gfCNCPoint4[3640] = {X 471.9427, Y 20.0094, Z -5.5000, A 0.000, B 0.000, C 0.000 }
gfCNCPoint4[3641] = {X 472.1592, Y 18.2535, Z -5.5000, A 0.000, B 0.000, C 0.000 }
gfCNCPoint4[3642] = {X 472.5540, Y 16.5288, Z -5.5000, A 0.000, B 0.000, C 0.000 }
gfCNCPoint4[3643] = {X 473.0727, Y 15.0578, Z -5.5000, A 0.000, B 0.000, C 0.000 }
gfCNCPoint4[3644] = {X 473.7721, Y 13.6637, Z -5.5000, A 0.000, B 0.000, C 0.000 }
gfCNCPoint4[3645] = {X 474.6410, Y 12.3684, Z -5.5000, A 0.000, B 0.000, C 0.000 }
gfCNCPoint4[3646] = {X 475.6658, Y 11.1925, Z -5.5000, A 0.000, B 0.000, C 0.000 }
gfCNCPoint4[3647] = {X 476.7434, Y 10.2234, Z -5.5000, A 0.000, B 0.000, C 0.000 }
gfCNCPoint4[3648] = {X 477.9268, Y 9.3867, Z -5.5000, A 0.000, B 0.000, C 0.000 }
gfCNCPoint4[3649] = {X 479.1997, Y 8.6938, Z -5.5000, A 0.000, B 0.000, C 0.000 }
gfCNCPoint4[3650] = {X 480.5449, Y 8.1544, Z -5.5000, A 0.000, B 0.000, C 0.000 }
gfCNCPoint4[3651] = {X 481.9438, Y 7.7756, Z -5.5000, A 0.000, B 0.000, C 0.000 }
gfCNCPoint4[3652] = {X 484.0949, Y 7.4404, Z -5.5000, A 0.000, B 0.000, C 0.000 }
gfCNCPoint4[3653] = {X 486.2687, Y 7.3224, Z -5.5000, A 0.000, B 0.000, C 0.000 }
gfCNCPoint4[3654] = {X 486.9707, Y 7.3102, Z -5.5000, A 0.000, B 0.000, C 0.000 }
gfCNCPoint4[3655] = {X 502.2122, Y 7.3103, Z -5.5000, A 0.000, B 0.000, C 0.000 }
gfCNCPoint4[3656] = {X 502.7439, Y 7.3144, Z -5.5000, A 0.000, B 0.000, C 0.000 }
gfCNCPoint4[3657] = {X 503.6982, Y 7.4166, Z -5.5000, A 0.000, B 0.000, C 0.000 }
gfCNCPoint4[3658] = {X 504.6139, Y 7.7042, Z -5.5000, A 0.000, B 0.000, C 0.000 }
gfCNCPoint4[3659] = {X 505.4552, Y 8.1661, Z -5.5000, A 0.000, B 0.000, C 0.000 }
gfCNCPoint4[3660] = {X 506.1895, Y 8.7843, Z -5.5000, A 0.000, B 0.000, C 0.000 }
gfCNCPoint4[3661] = {X 506.7880, Y 9.5346, Z -5.5000, A 0.000, B 0.000, C 0.000 }
gfCNCPoint4[3662] = {X 507.2274, Y 10.3879, Z -5.5000, A 0.000, B 0.000, C 0.000 }
gfCNCPoint4[3663] = {X 507.4825, Y 11.2663, Z -5.5000, A 0.000, B 0.000, C 0.000 }
gfCNCPoint4[3664] = {X 507.5685, Y 12.1769, Z -5.5000, A 0.000, B 0.000, C 0.000 }
gfCNCPoint4[3665] = {X 507.5683, Y 13.0237, Z -5.5000, A 0.000, B 0.000, C 0.000 }
gfCNCPoint4[3666] = {X 507.4609, Y 13.9970, Z -5.5000, A 0.000, B 0.000, C 0.000 }
gfCNCPoint4[3667] = {X 507.1614, Y 14.9292, Z -5.5000, A 0.000, B 0.000, C 0.000 }
gfCNCPoint4[3668] = {X 506.6818, Y 15.7829, Z -5.5000, A 0.000, B 0.000, C 0.000 }
gfCNCPoint4[3669] = {X 506.0415, Y 16.5237, Z -5.5000, A 0.000, B 0.000, C 0.000 }
gfCNCPoint4[3670] = {X 506.0414, Y 40.6631, Z -5.5000, A 0.000, B 0.000, C 0.000 }
gfCNCPoint4[3671] = {X 506.6823, Y 41.4045, Z -5.5000, A 0.000, B 0.000, C 0.000 }
gfCNCPoint4[3672] = {X 507.1621, Y 42.2591, Z -5.5000, A 0.000, B 0.000, C 0.000 }
gfCNCPoint4[3673] = {X 507.4614, Y 43.1923, Z -5.5000, A 0.000, B 0.000, C 0.000 }
gfCNCPoint4[3674] = {X 507.5683, Y 44.1665, Z -5.5000, A 0.000, B 0.000, C 0.000 }
gfCNCPoint4[3675] = {X 507.5685, Y 45.0000, Z -5.5000, A 0.000, B 0.000, C 0.000 }
gfCNCPoint4[3676] = {X 507.4747, Y 45.9520, Z -5.5000, A 0.000, B 0.000, C 0.000 }
gfCNCPoint4[3677] = {X 507.1970, Y 46.8675, Z -5.5000, A 0.000, B 0.000, C 0.000 }
gfCNCPoint4[3678] = {X 506.7461, Y 47.7112, Z -5.5000, A 0.000, B 0.000, C 0.000 }
gfCNCPoint4[3679] = {X 506.1392, Y 48.4507, Z -5.5000, A 0.000, B 0.000, C 0.000 }
gfCNCPoint4[3680] = {X 505.3997, Y 49.0576, Z -5.5000, A 0.000, B 0.000, C 0.000 }
gfCNCPoint4[3681] = {X 504.5560, Y 49.5085, Z -5.5000, A 0.000, B 0.000, C 0.000 }
gfCNCPoint4[3682] = {X 503.6405, Y 49.7862, Z -5.5000, A 0.000, B 0.000, C 0.000 }
gfCNCPoint4[3683] = {X 502.6885, Y 49.8800, Z -5.5000, A 0.000, B 0.000, C 0.000 }
gfCNCPoint4[3684] = {X 496.2450, Y 49.8800, Z -5.5000, A 0.000, B 0.000, C 0.000 }
gfCNCPoint4[3685] = {X 495.2220, Y 49.7716, Z -5.5000, A 0.000, B 0.000, C 0.000 }
gfCNCPoint4[3686] = {X 494.2445, Y 49.4511, Z -5.5000, A 0.000, B 0.000, C 0.000 }
gfCNCPoint4[3687] = {X 493.3559, Y 48.9328, Z -5.5000, A 0.000, B 0.000, C 0.000 }
gfCNCPoint4[3688] = {X 492.5956, Y 48.2398, Z -5.5000, A 0.000, B 0.000, C 0.000 }
gfCNCPoint4[3689] = {X 491.9976, Y 47.4028, Z -5.5000, A 0.000, B 0.000, C 0.000 }
gfCNCPoint4[3690] = {X 491.5882, Y 46.4590, Z -5.5000, A 0.000, B 0.000, C 0.000 }
gfCNCPoint4[3691] = {X 491.4241, Y 45.7570, Z -5.5000, A 0.000, B 0.000, C 0.000 }
gfCNCPoint4[3692] = {X 491.3652, Y 45.0385, Z -5.5000, A 0.000, B 0.000, C 0.000 }
gfCNCPoint4[3693] = {X 491.3655, Y 44.1416, Z -5.5000, A 0.000, B 0.000, C 0.000 }
gfCNCPoint4[3694] = {X 491.4758, Y 43.1751, Z -5.5000, A 0.000, B 0.000, C 0.000 }
gfCNCPoint4[3695] = {X 491.7756, Y 42.2497, Z -5.5000, A 0.000, B 0.000, C 0.000 }
gfCNCPoint4[3696] = {X 492.2530, Y 41.4020, Z -5.5000, A 0.000, B 0.000, C 0.000 }
gfCNCPoint4[3697] = {X 492.8890, Y 40.6660, Z -5.5000, A 0.000, B 0.000, C 0.000 }
gfCNCPoint4[3698] = {X 492.8890, Y 35.0338, Z -5.5000, A 0.000, B 0.000, C 0.000 }
gfCNCPoint4[3699] = {X 491.0668, Y 35.0338, Z -5.5000, A 0.000, B 0.000, C 0.000 }
gfCNCPoint4[3700] = {X 487.0440, Y 42.8709, Z -5.5000, A 0.000, B 0.000, C 0.000 }
gfCNCPoint4[3701] = {X 487.1810, Y 43.5116, Z -5.5000, A 0.000, B 0.000, C 0.000 }
gfCNCPoint4[3702] = {X 487.2308, Y 44.1648, Z -5.5000, A 0.000, B 0.000, C 0.000 }
gfCNCPoint4[3703] = {X 487.2310, Y 45.0000, Z -5.5000, A 0.000, B 0.000, C 0.000 }
gfCNCPoint4[3704] = {X 487.1749, Y 45.7380, Z -5.5000, A 0.000, B 0.000, C 0.000 }
gfCNCPoint4[3705] = {X 487.0078, Y 46.4590, Z -5.5000, A 0.000, B 0.000, C 0.000 }
gfCNCPoint4[3706] = {X 486.5939, Y 47.4110, Z -5.5000, A 0.000, B 0.000, C 0.000 }
gfCNCPoint4[3707] = {X 485.9879, Y 48.2538, Z -5.5000, A 0.000, B 0.000, C 0.000 }
gfCNCPoint4[3708] = {X 485.2175, Y 48.9494, Z -5.5000, A 0.000, B 0.000, C 0.000 }
gfCNCPoint4[3709] = {X 484.3173, Y 49.4663, Z -5.5000, A 0.000, B 0.000, C 0.000 }
gfCNCPoint4[3710] = {X 483.3557, Y 49.7755, Z -5.5000, A 0.000, B 0.000, C 0.000 }
gfCNCPoint4[3711] = {X 482.3510, Y 49.8800, Z -5.5000, A 0.000, B 0.000, C 0.000 }
gfCNCPoint4[3712] = {X 480.2695, Y 49.8800, Z -5.5000, A 0.000, B 0.000, C 0.000 }
gfCNCPoint4[3713] = {X 480.2695, Y 49.4000, Z -5.5000, A 0.000, B 0.000, C 0.000 }
gfCNCPoint4[3714] = {X 475.7650, Y 49.4000, Z -5.5000, A 0.000, B 0.000, C 0.000 }
gfCNCPoint4[3715] = {X 474.7859, Y 49.2897, Z -5.5000, A 0.000, B 0.000, C 0.000 }
gfCNCPoint4[3716] = {X 473.8559, Y 48.9643, Z -5.5000, A 0.000, B 0.000, C 0.000 }
gfCNCPoint4[3717] = {X 473.0216, Y 48.4401, Z -5.5000, A 0.000, B 0.000, C 0.000 }
gfCNCPoint4[3718] = {X 472.3249, Y 47.7434, Z -5.5000, A 0.000, B 0.000, C 0.000 }
gfCNCPoint4[3719] = {X 471.8007, Y 46.9091, Z -5.5000, A 0.000, B 0.000, C 0.000 }
gfCNCPoint4[3720] = {X 471.4753, Y 45.9791, Z -5.5000, A 0.000, B 0.000, C 0.000 }
gfCNCPoint4[3721] = {X 471.3650, Y 45.0000, Z -5.5000, A 0.000, B 0.000, C 0.000 }
gfCNCPoint4[3722] = {X 471.3654, Y 44.1483, Z -5.5000, A 0.000, B 0.000, C 0.000 }
gfCNCPoint4[3723] = {X 471.4638, Y 43.2816, Z -5.5000, A 0.000, B 0.000, C 0.000 }
gfCNCPoint4[3724] = {X 471.7311, Y 42.4514, Z -5.5000, A 0.000, B 0.000, C 0.000 }
gfCNCPoint4[3725] = {X 472.1570, Y 41.6903, Z -5.5000, A 0.000, B 0.000, C 0.000 }
gfCNCPoint4[3726] = {X 472.7247, Y 41.0281, Z -5.5000, A 0.000, B 0.000, C 0.000 }
gfCNCPoint4[3727] = {X 473.4118, Y 40.4909, Z -5.5000, A 0.000, B 0.000, C 0.000 }
gfCNCPoint4[3728] = {X 474.1914, Y 40.0998, Z -5.5000, A 0.000, B 0.000, C 0.000 }
gfCNCPoint4[3729] = {X 478.1276, Y 32.3950, Z -5.5000, A 0.000, B 0.000, C 0.000 }
gfCNCPoint4[3730] = {X 476.8703, Y 31.5214, Z -5.5000, A 0.000, B 0.000, C 0.000 }
gfCNCPoint4[3731] = {X 475.7398, Y 30.4889, Z -5.5000, A 0.000, B 0.000, C 0.000 }
gfCNCPoint4[3732] = {X 474.7559, Y 29.3158, Z -5.5000, A 0.000, B 0.000, C 0.000 }
gfCNCPoint4[3733] = {X 473.9361, Y 28.0227, Z -5.5000, A 0.000, B 0.000, C 0.000 }
gfCNCPoint4[3734] = {X 473.2948, Y 26.6325, Z -5.5000, A 0.000, B 0.000, C 0.000 }
gfCNCPoint4[3735] = {X 472.8433, Y 25.1695, Z -5.5000, A 0.000, B 0.000, C 0.000 }
gfCNCPoint4[3736] = {X 472.5277, Y 23.4784, Z -5.5000, A 0.000, B 0.000, C 0.000 }
gfCNCPoint4[3737] = {X 472.3866, Y 21.7639, Z -5.5000, A 0.000, B 0.000, C 0.000 }
gfCNCPoint4[3738] = {X 472.4215, Y 20.0440, Z -5.5000, A 0.000, B 0.000, C 0.000 }
gfCNCPoint4[3739] = {X 472.6320, Y 18.3366, Z -5.5000, A 0.000, B 0.000, C 0.000 }
gfCNCPoint4[3740] = {X 473.0158, Y 16.6597, Z -5.5000, A 0.000, B 0.000, C 0.000 }
gfCNCPoint4[3741] = {X 473.5624, Y 15.1345, Z -5.5000, A 0.000, B 0.000, C 0.000 }
gfCNCPoint4[3742] = {X 474.3108, Y 13.6976, Z -5.5000, A 0.000, B 0.000, C 0.000 }
gfCNCPoint4[3743] = {X 475.2472, Y 12.3756, Z -5.5000, A 0.000, B 0.000, C 0.000 }
gfCNCPoint4[3744] = {X 476.3545, Y 11.1928, Z -5.5000, A 0.000, B 0.000, C 0.000 }
gfCNCPoint4[3745] = {X 477.6119, Y 10.1712, Z -5.5000, A 0.000, B 0.000, C 0.000 }
gfCNCPoint4[3746] = {X 478.9964, Y 9.3297, Z -5.5000, A 0.000, B 0.000, C 0.000 }
gfCNCPoint4[3747] = {X 480.4822, Y 8.6838, Z -5.5000, A 0.000, B 0.000, C 0.000 }
gfCNCPoint4[3748] = {X 482.0419, Y 8.2455, Z -5.5000, A 0.000, B 0.000, C 0.000 }
gfCNCPoint4[3749] = {X 484.1468, Y 7.9175, Z -5.5000, A 0.000, B 0.000, C 0.000 }
gfCNCPoint4[3750] = {X 486.2739, Y 7.8024, Z -5.5000, A 0.000, B 0.000, C 0.000 }
gfCNCPoint4[3751] = {X 486.9707, Y 7.7902, Z -5.5000, A 0.000, B 0.000, C 0.000 }
gfCNCPoint4[3752] = {X 502.2084, Y 7.7902, Z -5.5000, A 0.000, B 0.000, C 0.000 }
gfCNCPoint4[3753] = {X 502.7401, Y 7.7944, Z -5.5000, A 0.000, B 0.000, C 0.000 }
gfCNCPoint4[3754] = {X 503.7097, Y 7.9108, Z -5.5000, A 0.000, B 0.000, C 0.000 }
gfCNCPoint4[3755] = {X 504.6294, Y 8.2389, Z -5.5000, A 0.000, B 0.000, C 0.000 }
gfCNCPoint4[3756] = {X 505.4537, Y 8.7626, Z -5.5000, A 0.000, B 0.000, C 0.000 }
gfCNCPoint4[3757] = {X 506.1415, Y 9.4558, Z -5.5000, A 0.000, B 0.000, C 0.000 }
gfCNCPoint4[3758] = {X 506.6587, Y 10.2841, Z -5.5000, A 0.000, B 0.000, C 0.000 }
gfCNCPoint4[3759] = {X 506.9797, Y 11.2064, Z -5.5000, A 0.000, B 0.000, C 0.000 }
gfCNCPoint4[3760] = {X 507.0885, Y 12.1769, Z -5.5000, A 0.000, B 0.000, C 0.000 }
gfCNCPoint4[3761] = {X 507.0883, Y 13.0233, Z -5.5000, A 0.000, B 0.000, C 0.000 }
gfCNCPoint4[3762] = {X 506.9800, Y 13.9492, Z -5.5000, A 0.000, B 0.000, C 0.000 }
gfCNCPoint4[3763] = {X 506.6791, Y 14.8314, Z -5.5000, A 0.000, B 0.000, C 0.000 }
gfCNCPoint4[3764] = {X 506.1991, Y 15.6305, Z -5.5000, A 0.000, B 0.000, C 0.000 }
gfCNCPoint4[3765] = {X 505.5615, Y 16.3106, Z -5.5000, A 0.000, B 0.000, C 0.000 }
gfCNCPoint4[3766] = {X 505.5614, Y 40.8762, Z -5.5000, A 0.000, B 0.000, C 0.000 }
gfCNCPoint4[3767] = {X 506.2059, Y 41.5653, Z -5.5000, A 0.000, B 0.000, C 0.000 }
gfCNCPoint4[3768] = {X 506.6886, Y 42.3759, Z -5.5000, A 0.000, B 0.000, C 0.000 }
gfCNCPoint4[3769] = {X 506.9874, Y 43.2708, Z -5.5000, A 0.000, B 0.000, C 0.000 }
gfCNCPoint4[3770] = {X 507.0885, Y 44.2089, Z -5.5000, A 0.000, B 0.000, C 0.000 }
gfCNCPoint4[3771] = {X 507.0885, Y 45.0000, Z -5.5000, A 0.000, B 0.000, C 0.000 }
gfCNCPoint4[3772] = {X 506.9782, Y 45.9791, Z -5.5000, A 0.000, B 0.000, C 0.000 }
gfCNCPoint4[3773] = {X 506.6528, Y 46.9091, Z -5.5000, A 0.000, B 0.000, C 0.000 }
gfCNCPoint4[3774] = {X 506.1285, Y 47.7434, Z -5.5000, A 0.000, B 0.000, C 0.000 }
gfCNCPoint4[3775] = {X 505.4318, Y 48.4401, Z -5.5000, A 0.000, B 0.000, C 0.000 }
gfCNCPoint4[3776] = {X 504.5976, Y 48.9643, Z -5.5000, A 0.000, B 0.000, C 0.000 }
gfCNCPoint4[3777] = {X 503.6676, Y 49.2897, Z -5.5000, A 0.000, B 0.000, C 0.000 }
gfCNCPoint4[3778] = {X 502.6885, Y 49.4000, Z -5.5000, A 0.000, B 0.000, C 0.000 }
gfCNCPoint4[3779] = {X 496.2450, Y 49.4000, Z -5.5000, A 0.000, B 0.000, C 0.000 }
gfCNCPoint4[3780] = {X 495.2659, Y 49.2897, Z -5.5000, A 0.000, B 0.000, C 0.000 }
gfCNCPoint4[3781] = {X 494.3359, Y 48.9643, Z -5.5000, A 0.000, B 0.000, C 0.000 }
gfCNCPoint4[3782] = {X 493.5017, Y 48.4400, Z -5.5000, A 0.000, B 0.000, C 0.000 }
gfCNCPoint4[3783] = {X 492.8050, Y 47.7433, Z -5.5000, A 0.000, B 0.000, C 0.000 }
gfCNCPoint4[3784] = {X 492.2808, Y 46.9091, Z -5.5000, A 0.000, B 0.000, C 0.000 }
gfCNCPoint4[3785] = {X 491.9553, Y 45.9791, Z -5.5000, A 0.000, B 0.000, C 0.000 }
gfCNCPoint4[3786] = {X 491.8450, Y 45.0000, Z -5.5000, A 0.000, B 0.000, C 0.000 }
gfCNCPoint4[3787] = {X 491.8454, Y 44.1483, Z -5.5000, A 0.000, B 0.000, C 0.000 }
gfCNCPoint4[3788] = {X 491.9559, Y 43.2275, Z -5.5000, A 0.000, B 0.000, C 0.000 }
gfCNCPoint4[3789] = {X 492.2568, Y 42.3503, Z -5.5000, A 0.000, B 0.000, C 0.000 }
gfCNCPoint4[3790] = {X 492.7349, Y 41.5556, Z -5.5000, A 0.000, B 0.000, C 0.000 }
gfCNCPoint4[3791] = {X 493.3690, Y 40.8789, Z -5.5000, A 0.000, B 0.000, C 0.000 }
gfCNCPoint4[3792] = {X 493.3690, Y 34.5538, Z -5.5000, A 0.000, B 0.000, C 0.000 }
gfCNCPoint4[3793] = {X 490.7737, Y 34.5538, Z -5.5000, A 0.000, B 0.000, C 0.000 }
gfCNCPoint4[3794] = {X 486.6332, Y 42.6204, Z -5.5000, A 0.000, B 0.000, C 0.000 }
gfCNCPoint4[3795] = {X 486.5275, Y 42.8242, Z -5.5000, A 0.000, B 0.000, C 0.000 }
gfCNCPoint4[3796] = {X 486.6948, Y 43.5076, Z -5.5000, A 0.000, B 0.000, C 0.000 }
gfCNCPoint4[3797] = {X 486.7510, Y 44.2089, Z -5.5000, A 0.000, B 0.000, C 0.000 }
gfCNCPoint4[3798] = {X 486.7510, Y 45.0000, Z -5.5000, A 0.000, B 0.000, C 0.000 }
gfCNCPoint4[3799] = {X 486.6407, Y 45.9791, Z -5.5000, A 0.000, B 0.000, C 0.000 }
gfCNCPoint4[3800] = {X 486.3153, Y 46.9091, Z -5.5000, A 0.000, B 0.000, C 0.000 }
gfCNCPoint4[3801] = {X 485.7911, Y 47.7434, Z -5.5000, A 0.000, B 0.000, C 0.000 }
gfCNCPoint4[3802] = {X 485.0944, Y 48.4401, Z -5.5000, A 0.000, B 0.000, C 0.000 }
gfCNCPoint4[3803] = {X 484.2601, Y 48.9643, Z -5.5000, A 0.000, B 0.000, C 0.000 }
gfCNCPoint4[3804] = {X 483.3301, Y 49.2897, Z -5.5000, A 0.000, B 0.000, C 0.000 }
gfCNCPoint4[3805] = {X 482.3510, Y 49.4000, Z -5.5000, A 0.000, B 0.000, C 0.000 }
gfCNCPoint4[3806] = {X 480.2695, Y 49.4000, Z -5.5000, A 0.000, B 0.000, C 0.000 }
gfCNCPoint4[3807] = {X 480.2695, Y 49.8800, Z -5.5000, A 0.000, B 0.000, C 0.000 }
gfCNCPoint4[3808] = {X 481.4067, Y 50.7435, Z -5.5000, A 0.000, B 0.000, C 0.000 }
gfCNCPoint4[3809] = {X 482.4044, Y 51.7649, Z -5.5000, A 0.000, B 0.000, C 0.000 }
gfCNCPoint4[3810] = {X 483.2411, Y 52.9219, Z -5.5000, A 0.000, B 0.000, C 0.000 }
gfCNCPoint4[3811] = {X 483.8615, Y 54.1044, Z -5.5000, A 0.000, B 0.000, C 0.000 }
gfCNCPoint4[3812] = {X 484.3133, Y 55.3610, Z -5.5000, A 0.000, B 0.000, C 0.000 }
gfCNCPoint4[3813] = {X 484.5879, Y 56.6678, Z -5.5000, A 0.000, B 0.000, C 0.000 }
gfCNCPoint4[3814] = {X 484.6800, Y 58.0000, Z -5.5000, A 0.000, B 0.000, C 0.000 }
gfCNCPoint4[3815] = {X 484.6797, Y 59.0140, Z -5.5000, A 0.000, B 0.000, C 0.000 }
gfCNCPoint4[3816] = {X 484.5592, Y 60.4584, Z -5.5000, A 0.000, B 0.000, C 0.000 }
gfCNCPoint4[3817] = {X 484.2245, Y 61.8685, Z -5.5000, A 0.000, B 0.000, C 0.000 }
gfCNCPoint4[3818] = {X 483.6830, Y 63.2129, Z -5.5000, A 0.000, B 0.000, C 0.000 }
gfCNCPoint4[3819] = {X 482.9468, Y 64.4613, Z -5.5000, A 0.000, B 0.000, C 0.000 }
gfCNCPoint4[3820] = {X 482.0325, Y 65.5859, Z -5.5000, A 0.000, B 0.000, C 0.000 }
gfCNCPoint4[3821] = {X 480.9605, Y 66.5613, Z -5.5000, A 0.000, B 0.000, C 0.000 }
gfCNCPoint4[3822] = {X 480.9609, Y 89.4440, Z -5.5000, A 0.000, B 0.000, C 0.000 }
gfCNCPoint4[3823] = {X 482.0606, Y 90.4464, Z -5.5000, A 0.000, B 0.000, C 0.000 }
gfCNCPoint4[3824] = {X 482.9931, Y 91.6060, Z -5.5000, A 0.000, B 0.000, C 0.000 }
gfCNCPoint4[3825] = {X 483.7364, Y 92.8951, Z -5.5000, A 0.000, B 0.000, C 0.000 }
gfCNCPoint4[3826] = {X 507.6814, Y 92.8951, Z -5.5000, A 0.000, B 0.000, C 0.000 }
gfCNCPoint4[3827] = {X 507.6814, Y 95.2951, Z -5.5000, A 0.000, B 0.000, C 0.000 }
gfCNCPoint4[3828] = {X 595.2966, Y 95.2951, Z -5.5000, A 0.000, B 0.000, C 0.000 }
gfCNCPoint4[3829] = {X 595.2966, Y 54.2000, Z -5.5000, A 0.000, B 0.000, C 0.000 }
gfCNCPoint4[3830] = {X 593.5565, Y 54.2000, Z -5.5000, A 0.000, B 0.000, C 0.000 }
gfCNCPoint4[3831] = {X 592.2403, Y 54.1053, Z -5.5000, A 0.000, B 0.000, C 0.000 }
gfCNCPoint4[3832] = {X 590.9511, Y 53.8233, Z -5.5000, A 0.000, B 0.000, C 0.000 }
gfCNCPoint4[3833] = {X 589.7155, Y 53.3598, Z -5.5000, A 0.000, B 0.000, C 0.000 }
gfCNCPoint4[3834] = {X 588.5589, Y 52.7242, Z -5.5000, A 0.000, B 0.000, C 0.000 }
gfCNCPoint4[3835] = {X 587.5052, Y 51.9297, Z -5.5000, A 0.000, B 0.000, C 0.000 }
gfCNCPoint4[3836] = {X 586.4956, Y 52.6955, Z -5.5000, A 0.000, B 0.000, C 0.000 }
gfCNCPoint4[3837] = {X 585.3903, Y 53.3153, Z -5.5000, A 0.000, B 0.000, C 0.000 }
gfCNCPoint4[3838] = {X 584.1375, Y 53.7999, Z -5.5000, A 0.000, B 0.000, C 0.000 }
gfCNCPoint4[3839] = {X 582.8276, Y 54.0969, Z -5.5000, A 0.000, B 0.000, C 0.000 }
gfCNCPoint4[3840] = {X 581.4884, Y 54.1999, Z -5.5000, A 0.000, B 0.000, C 0.000 }
gfCNCPoint4[3841] = {X 580.1485, Y 54.1069, Z -5.5000, A 0.000, B 0.000, C 0.000 }
gfCNCPoint4[3842] = {X 578.8364, Y 53.8198, Z -5.5000, A 0.000, B 0.000, C 0.000 }
gfCNCPoint4[3843] = {X 577.5801, Y 53.3447, Z -5.5000, A 0.000, B 0.000, C 0.000 }
gfCNCPoint4[3844] = {X 576.4063, Y 52.6917, Z -5.5000, A 0.000, B 0.000, C 0.000 }
gfCNCPoint4[3845] = {X 575.3401, Y 51.8748, Z -5.5000, A 0.000, B 0.000, C 0.000 }
gfCNCPoint4[3846] = {X 574.2798, Y 52.6879, Z -5.5000, A 0.000, B 0.000, C 0.000 }
gfCNCPoint4[3847] = {X 573.1128, Y 53.3388, Z -5.5000, A 0.000, B 0.000, C 0.000 }
gfCNCPoint4[3848] = {X 571.8638, Y 53.8139, Z -5.5000, A 0.000, B 0.000, C 0.000 }
gfCNCPoint4[3849] = {X 570.5592, Y 54.1030, Z -5.5000, A 0.000, B 0.000, C 0.000 }
gfCNCPoint4[3850] = {X 569.2264, Y 54.2000, Z -5.5000, A 0.000, B 0.000, C 0.000 }
gfCNCPoint4[3851] = {X 562.4443, Y 54.2000, Z -5.5000, A 0.000, B 0.000, C 0.000 }
gfCNCPoint4[3852] = {X 561.0051, Y 54.0867, Z -5.5000, A 0.000, B 0.000, C 0.000 }
gfCNCPoint4[3853] = {X 559.6013, Y 53.7497, Z -5.5000, A 0.000, B 0.000, C 0.000 }
gfCNCPoint4[3854] = {X 558.2676, Y 53.1973, Z -5.5000, A 0.000, B 0.000, C 0.000 }
gfCNCPoint4[3855] = {X 557.0367, Y 52.4430, Z -5.5000, A 0.000, B 0.000, C 0.000 }
gfCNCPoint4[3856] = {X 555.9389, Y 51.5054, Z -5.5000, A 0.000, B 0.000, C 0.000 }
gfCNCPoint4[3857] = {X 555.0013, Y 50.4076, Z -5.5000, A 0.000, B 0.000, C 0.000 }
gfCNCPoint4[3858] = {X 554.2470, Y 49.1767, Z -5.5000, A 0.000, B 0.000, C 0.000 }
gfCNCPoint4[3859] = {X 553.6946, Y 47.8430, Z -5.5000, A 0.000, B 0.000, C 0.000 }
gfCNCPoint4[3860] = {X 553.3576, Y 46.4392, Z -5.5000, A 0.000, B 0.000, C 0.000 }
gfCNCPoint4[3861] = {X 553.2443, Y 45.0000, Z -5.5000, A 0.000, B 0.000, C 0.000 }
gfCNCPoint4[3862] = {X 553.2443, Y 44.0608, Z -5.5000, A 0.000, B 0.000, C 0.000 }
gfCNCPoint4[3863] = {X 553.3446, Y 42.7243, Z -5.5000, A 0.000, B 0.000, C 0.000 }
gfCNCPoint4[3864] = {X 553.6373, Y 41.4165, Z -5.5000, A 0.000, B 0.000, C 0.000 }
gfCNCPoint4[3865] = {X 554.1163, Y 40.1648, Z -5.5000, A 0.000, B 0.000, C 0.000 }
gfCNCPoint4[3866] = {X 554.7715, Y 38.9956, Z -5.5000, A 0.000, B 0.000, C 0.000 }
gfCNCPoint4[3867] = {X 554.7715, Y 11.0103, Z -5.5000, A 0.000, B 0.000, C 0.000 }
gfCNCPoint4[3868] = {X 554.1216, Y 9.8549, Z -5.5000, A 0.000, B 0.000, C 0.000 }
gfCNCPoint4[3869] = {X 553.6445, Y 8.6181, Z -5.5000, A 0.000, B 0.000, C 0.000 }
gfCNCPoint4[3870] = {X 553.3502, Y 7.3257, Z -5.5000, A 0.000, B 0.000, C 0.000 }
gfCNCPoint4[3871] = {X 553.2446, Y 6.0043, Z -5.5000, A 0.000, B 0.000, C 0.000 }
gfCNCPoint4[3872] = {X 553.2443, Y 5.0000, Z -5.5000, A 0.000, B 0.000, C 0.000 }
gfCNCPoint4[3873] = {X 553.2455, Y 4.8524, Z -5.5000, A 0.000, B 0.000, C 0.000 }
gfCNCPoint4[3874] = {X 553.2490, Y 4.7049, Z -5.5000, A 0.000, B 0.000, C 0.000 }
gfCNCPoint4[3875] = {X 365.1876, Y 4.7049, Z -5.5000, A 0.000, B 0.000, C 0.000 }
gfCNCPoint4[3876] = {X 365.6156, Y 5.1720, Z -5.5000, A 0.000, B 0.000, C 0.000 }
gfCNCPoint4[3877] = {X 366.0311, Y 5.6503, Z -5.5000, A 0.000, B 0.000, C 0.000 }
gfCNCPoint4[3878] = {X 367.1000, Y 7.0011, Z -5.5000, A 0.000, B 0.000, C 0.000 }
gfCNCPoint4[3879] = {X 368.0841, Y 8.4149, Z -5.5000, A 0.000, B 0.000, C 0.000 }
gfCNCPoint4[3880] = {X 369.2514, Y 10.3772, Z -5.5000, A 0.000, B 0.000, C 0.000 }
gfCNCPoint4[3881] = {X 370.2554, Y 12.4279, Z -5.5000, A 0.000, B 0.000, C 0.000 }
gfCNCPoint4[3882] = {X 371.0892, Y 14.5535, Z -5.5000, A 0.000, B 0.000, C 0.000 }
gfCNCPoint4[3883] = {X 371.7476, Y 16.7398, Z -5.5000, A 0.000, B 0.000, C 0.000 }
gfCNCPoint4[3884] = {X 372.2259, Y 18.9724, Z -5.5000, A 0.000, B 0.000, C 0.000 }
gfCNCPoint4[3885] = {X 372.5706, Y 21.4029, Z -5.5000, A 0.000, B 0.000, C 0.000 }
gfCNCPoint4[3886] = {X 372.7426, Y 23.8518, Z -5.5000, A 0.000, B 0.000, C 0.000 }
gfCNCPoint4[3887] = {X 372.7409, Y 26.3067, Z -5.5000, A 0.000, B 0.000, C 0.000 }
gfCNCPoint4[3888] = {X 372.5657, Y 28.7553, Z -5.5000, A 0.000, B 0.000, C 0.000 }
gfCNCPoint4[3889] = {X 372.2177, Y 31.1854, Z -5.5000, A 0.000, B 0.000, C 0.000 }
gfCNCPoint4[3890] = {X 371.7664, Y 33.2924, Z -5.5000, A 0.000, B 0.000, C 0.000 }
gfCNCPoint4[3891] = {X 371.1518, Y 35.3577, Z -5.5000, A 0.000, B 0.000, C 0.000 }
gfCNCPoint4[3892] = {X 370.3777, Y 37.3687, Z -5.5000, A 0.000, B 0.000, C 0.000 }
gfCNCPoint4[3893] = {X 369.4488, Y 39.3130, Z -5.5000, A 0.000, B 0.000, C 0.000 }
gfCNCPoint4[3894] = {X 368.3708, Y 41.1787, Z -5.5000, A 0.000, B 0.000, C 0.000 }
gfCNCPoint4[3895] = {X 367.1502, Y 42.9545, Z -5.5000, A 0.000, B 0.000, C 0.000 }
gfCNCPoint4[3896] = {X 365.8288, Y 44.5908, Z -5.5000, A 0.000, B 0.000, C 0.000 }
gfCNCPoint4[3897] = {X 364.3743, Y 46.1099, Z -5.5000, A 0.000, B 0.000, C 0.000 }
gfCNCPoint4[3898] = {X 362.7969, Y 47.5011, Z -5.5000, A 0.000, B 0.000, C 0.000 }
gfCNCPoint4[3899] = {X 361.1080, Y 48.7545, Z -5.5000, A 0.000, B 0.000, C 0.000 }
gfCNCPoint4[3900] = {X 359.3195, Y 49.8611, Z -5.5000, A 0.000, B 0.000, C 0.000 }
gfCNCPoint4[3901] = {X 357.4441, Y 50.8132, Z -5.5000, A 0.000, B 0.000, C 0.000 }
gfCNCPoint4[3902] = {X 355.4664, Y 51.5790, Z -5.5000, A 0.000, B 0.000, C 0.000 }
gfCNCPoint4[3903] = {X 353.4327, Y 52.1809, Z -5.5000, A 0.000, B 0.000, C 0.000 }
gfCNCPoint4[3904] = {X 351.3568, Y 52.6150, Z -5.5000, A 0.000, B 0.000, C 0.000 }
gfCNCPoint4[3905] = {X 349.2523, Y 52.8783, Z -5.5000, A 0.000, B 0.000, C 0.000 }
gfCNCPoint4[3906] = {X 347.1334, Y 52.9692, Z -5.5000, A 0.000, B 0.000, C 0.000 }
gfCNCPoint4[3907] = {X 344.8132, Y 52.9269, Z -5.5000, A 0.000, B 0.000, C 0.000 }
gfCNCPoint4[3908] = {X 342.5054, Y 52.6838, Z -5.5000, A 0.000, B 0.000, C 0.000 }
gfCNCPoint4[3909] = {X 340.2273, Y 52.2417, Z -5.5000, A 0.000, B 0.000, C 0.000 }
gfCNCPoint4[3910] = {X 337.9960, Y 51.6040, Z -5.5000, A 0.000, B 0.000, C 0.000 }
gfCNCPoint4[3911] = {X 335.8284, Y 50.7754, Z -5.5000, A 0.000, B 0.000, C 0.000 }
gfCNCPoint4[3912] = {X 333.7407, Y 49.7622, Z -5.5000, A 0.000, B 0.000, C 0.000 }
gfCNCPoint4[3913] = {X 332.8368, Y 49.2304, Z -5.5000, A 0.000, B 0.000, C 0.000 }
gfCNCPoint4[3914] = {X 331.9545, Y 48.6635, Z -5.5000, A 0.000, B 0.000, C 0.000 }
gfCNCPoint4[3915] = {X 331.3029, Y 48.2124, Z -5.5000, A 0.000, B 0.000, C 0.000 }
gfCNCPoint4[3916] = {X 330.6649, Y 47.7422, Z -5.5000, A 0.000, B 0.000, C 0.000 }
gfCNCPoint4[3917] = {X 329.2125, Y 49.6529, Z -5.5000, A 0.000, B 0.000, C 0.000 }
gfCNCPoint4[3918] = {X 328.8696, Y 49.3882, Z -5.5000, A 0.000, B 0.000, C 0.000 }
gfCNCPoint4[3919] = {X 328.5307, Y 49.1184, Z -5.5000, A 0.000, B 0.000, C 0.000 }
gfCNCPoint4[3920] = {X 328.1261, Y 49.0389, Z -5.5000, A 0.000, B 0.000, C 0.000 }
gfCNCPoint4[3921] = {X 327.7253, Y 48.9423, Z -5.5000, A 0.000, B 0.000, C 0.000 }
gfCNCPoint4[3922] = {X 328.4841, Y 49.2659, Z -5.5000, A 0.000, B 0.000, C 0.000 }
gfCNCPoint4[3923] = {X 329.2125, Y 49.6529, Z -5.5000, A 0.000, B 0.000, C 0.000 }
gfCNCPoint4[3924] = {X 330.6649, Y 47.7422, Z -5.5000, A 0.000, B 0.000, C 0.000 }
gfCNCPoint4[3925] = {X 330.0928, Y 47.2950, Z -5.5000, A 0.000, B 0.000, C 0.000 }
gfCNCPoint4[3926] = {X 329.5331, Y 46.8323, Z -5.5000, A 0.000, B 0.000, C 0.000 }
gfCNCPoint4[3927] = {X 328.9309, Y 46.7519, Z -5.5000, A 0.000, B 0.000, C 0.000 }
gfCNCPoint4[3928] = {X 328.3374, Y 46.6216, Z -5.5000, A 0.000, B 0.000, C 0.000 }
gfCNCPoint4[3929] = {X 327.9789, Y 46.5172, Z -5.5000, A 0.000, B 0.000, C 0.000 }
gfCNCPoint4[3930] = {X 327.6263, Y 46.3944, Z -5.5000, A 0.000, B 0.000, C 0.000 }
gfCNCPoint4[3931] = {X 326.7320, Y 45.9864, Z -5.5000, A 0.000, B 0.000, C 0.000 }
gfCNCPoint4[3932] = {X 325.9009, Y 45.4616, Z -5.5000, A 0.000, B 0.000, C 0.000 }
gfCNCPoint4[3933] = {X 325.1480, Y 44.8296, Z -5.5000, A 0.000, B 0.000, C 0.000 }
gfCNCPoint4[3934] = {X 324.5140, Y 44.2115, Z -5.5000, A 0.000, B 0.000, C 0.000 }
gfCNCPoint4[3935] = {X 324.0475, Y 43.7117, Z -5.5000, A 0.000, B 0.000, C 0.000 }
gfCNCPoint4[3936] = {X 323.6300, Y 43.1703, Z -5.5000, A 0.000, B 0.000, C 0.000 }
gfCNCPoint4[3937] = {X 319.6957, Y 45.9200, Z -5.5000, A 0.000, B 0.000, C 0.000 }
gfCNCPoint4[3938] = {X 319.4780, Y 45.5976, Z -5.5000, A 0.000, B 0.000, C 0.000 }
gfCNCPoint4[3939] = {X 319.2708, Y 45.2683, Z -5.5000, A 0.000, B 0.000, C 0.000 }
gfCNCPoint4[3940] = {X 319.2514, Y 45.5948, Z -5.5000, A 0.000, B 0.000, C 0.000 }
gfCNCPoint4[3941] = {X 319.2174, Y 45.9200, Z -5.5000, A 0.000, B 0.000, C 0.000 }
gfCNCPoint4[3942] = {X 319.6957, Y 45.9200, Z -5.5000, A 0.000, B 0.000, C 0.000 }
gfCNCPoint4[3943] = {X 321.6628, Y 44.5452, Z -5.5000, A 0.000, B 0.000, C 0.000 }
gfCNCPoint4[3944] = {X 321.4884, Y 44.2868, Z -5.5000, A 0.000, B 0.000, C 0.000 }
gfCNCPoint4[3945] = {X 321.3224, Y 44.0230, Z -5.5000, A 0.000, B 0.000, C 0.000 }
gfCNCPoint4[3946] = {X 320.6709, Y 42.7450, Z -5.5000, A 0.000, B 0.000, C 0.000 }
gfCNCPoint4[3947] = {X 320.2155, Y 41.3847, Z -5.5000, A 0.000, B 0.000, C 0.000 }
gfCNCPoint4[3948] = {X 319.9661, Y 39.9721, Z -5.5000, A 0.000, B 0.000, C 0.000 }
gfCNCPoint4[3949] = {X 319.9282, Y 38.5381, Z -5.5000, A 0.000, B 0.000, C 0.000 }
gfCNCPoint4[3950] = {X 320.1026, Y 37.1143, Z -5.5000, A 0.000, B 0.000, C 0.000 }
gfCNCPoint4[3951] = {X 320.4307, Y 35.8890, Z -5.5000, A 0.000, B 0.000, C 0.000 }
gfCNCPoint4[3952] = {X 320.9162, Y 34.7170, Z -5.5000, A 0.000, B 0.000, C 0.000 }
gfCNCPoint4[3953] = {X 321.5508, Y 33.6186, Z -5.5000, A 0.000, B 0.000, C 0.000 }
gfCNCPoint4[3954] = {X 324.1389, Y 29.7489, Z -5.5000, A 0.000, B 0.000, C 0.000 }
gfCNCPoint4[3955] = {X 320.1490, Y 27.0804, Z -5.5000, A 0.000, B 0.000, C 0.000 }
gfCNCPoint4[3956] = {X 321.8041, Y 24.6058, Z -5.5000, A 0.000, B 0.000, C 0.000 }
gfCNCPoint4[3957] = {X 321.9897, Y 24.3356, Z -5.5000, A 0.000, B 0.000, C 0.000 }
gfCNCPoint4[3958] = {X 322.1814, Y 24.0697, Z -5.5000, A 0.000, B 0.000, C 0.000 }
gfCNCPoint4[3959] = {X 321.5380, Y 23.0772, Z -5.5000, A 0.000, B 0.000, C 0.000 }
gfCNCPoint4[3960] = {X 320.9777, Y 22.0354, Z -5.5000, A 0.000, B 0.000, C 0.000 }
gfCNCPoint4[3961] = {X 320.1493, Y 20.3314, Z -5.5000, A 0.000, B 0.000, C 0.000 }
gfCNCPoint4[3962] = {X 320.1490, Y 27.0804, Z -5.5000, A 0.000, B 0.000, C 0.000 }
gfCNCPoint4[3963] = {X 322.1440, Y 28.4147, Z -5.5000, A 0.000, B 0.000, C 0.000 }
gfCNCPoint4[3964] = {X 323.7974, Y 25.9424, Z -5.5000, A 0.000, B 0.000, C 0.000 }
gfCNCPoint4[3965] = {X 324.5112, Y 24.9841, Z -5.5000, A 0.000, B 0.000, C 0.000 }
gfCNCPoint4[3966] = {X 325.3162, Y 24.1010, Z -5.5000, A 0.000, B 0.000, C 0.000 }
gfCNCPoint4[3967] = {X 324.4812, Y 23.1413, Z -5.5000, A 0.000, B 0.000, C 0.000 }
gfCNCPoint4[3968] = {X 323.7518, Y 22.0990, Z -5.5000, A 0.000, B 0.000, C 0.000 }
gfCNCPoint4[3969] = {X 323.1360, Y 20.9859, Z -5.5000, A 0.000, B 0.000, C 0.000 }
gfCNCPoint4[3970] = {X 319.6151, Y 13.7428, Z -5.5000, A 0.000, B 0.000, C 0.000 }
gfCNCPoint4[3971] = {X 319.4387, Y 13.3633, Z -5.5000, A 0.000, B 0.000, C 0.000 }
gfCNCPoint4[3972] = {X 319.2755, Y 12.9779, Z -5.5000, A 0.000, B 0.000, C 0.000 }
gfCNCPoint4[3973] = {X 319.2755, Y 13.0353, Z -5.5000, A 0.000, B 0.000, C 0.000 }
gfCNCPoint4[3974] = {X 319.1698, Y 14.2151, Z -5.5000, A 0.000, B 0.000, C 0.000 }
gfCNCPoint4[3975] = {X 318.8743, Y 15.3621, Z -5.5000, A 0.000, B 0.000, C 0.000 }
gfCNCPoint4[3976] = {X 318.3966, Y 16.4460, Z -5.5000, A 0.000, B 0.000, C 0.000 }
gfCNCPoint4[3977] = {X 317.7495, Y 17.4382, Z -5.5000, A 0.000, B 0.000, C 0.000 }
gfCNCPoint4[3978] = {X 317.7486, Y 36.6468, Z -5.5000, A 0.000, B 0.000, C 0.000 }
gfCNCPoint4[3979] = {X 318.1580, Y 35.1176, Z -5.5000, A 0.000, B 0.000, C 0.000 }
gfCNCPoint4[3980] = {X 318.7639, Y 33.6551, Z -5.5000, A 0.000, B 0.000, C 0.000 }
gfCNCPoint4[3981] = {X 319.5559, Y 32.2844, Z -5.5000, A 0.000, B 0.000, C 0.000 }
gfCNCPoint4[3982] = {X 322.1440, Y 28.4147, Z -5.5000, A 0.000, B 0.000, C 0.000 }
gfCNCPoint4[3983] = {X 324.1389, Y 29.7489, Z -5.5000, A 0.000, B 0.000, C 0.000 }
gfCNCPoint4[3984] = {X 325.7907, Y 27.2791, Z -5.5000, A 0.000, B 0.000, C 0.000 }
gfCNCPoint4[3985] = {X 326.3627, Y 26.5112, Z -5.5000, A 0.000, B 0.000, C 0.000 }
gfCNCPoint4[3986] = {X 327.0077, Y 25.8035, Z -5.5000, A 0.000, B 0.000, C 0.000 }
gfCNCPoint4[3987] = {X 328.0707, Y 24.8904, Z -5.5000, A 0.000, B 0.000, C 0.000 }
gfCNCPoint4[3988] = {X 329.2543, Y 24.1403, Z -5.5000, A 0.000, B 0.000, C 0.000 }
gfCNCPoint4[3989] = {X 328.0859, Y 23.3667, Z -5.5000, A 0.000, B 0.000, C 0.000 }
gfCNCPoint4[3990] = {X 327.0414, Y 22.4326, Z -5.5000, A 0.000, B 0.000, C 0.000 }
gfCNCPoint4[3991] = {X 326.3723, Y 21.6635, Z -5.5000, A 0.000, B 0.000, C 0.000 }
gfCNCPoint4[3992] = {X 325.7878, Y 20.8284, Z -5.5000, A 0.000, B 0.000, C 0.000 }
gfCNCPoint4[3993] = {X 325.2944, Y 19.9364, Z -5.5000, A 0.000, B 0.000, C 0.000 }
gfCNCPoint4[3994] = {X 321.7736, Y 12.6936, Z -5.5000, A 0.000, B 0.000, C 0.000 }
gfCNCPoint4[3995] = {X 321.6322, Y 12.3894, Z -5.5000, A 0.000, B 0.000, C 0.000 }
gfCNCPoint4[3996] = {X 321.5015, Y 12.0806, Z -5.5000, A 0.000, B 0.000, C 0.000 }
gfCNCPoint4[3997] = {X 321.1058, Y 10.8773, Z -5.5000, A 0.000, B 0.000, C 0.000 }
gfCNCPoint4[3998] = {X 320.8706, Y 9.6327, Z -5.5000, A 0.000, B 0.000, C 0.000 }
gfCNCPoint4[3999] = {X 320.7999, Y 8.3680, Z -5.5000, A 0.000, B 0.000, C 0.000 }
gfCNCPoint4[4000] = {X 320.8950, Y 7.1049, Z -5.5000, A 0.000, B 0.000, C 0.000 }
gfCNCPoint4[4001] = {X 298.7842, Y 7.1049, Z -5.5000, A 0.000, B 0.000, C 0.000 }
gfCNCPoint4[4002] = {X 298.7842, Y 9.5049, Z -5.5000, A 0.000, B 0.000, C 0.000 }
gfCNCPoint4[4003] = {X 297.8291, Y 9.5049, Z -5.5000, A 0.000, B 0.000, C 0.000 }
gfCNCPoint4[4004] = {X 298.1371, Y 10.4755, Z -5.5000, A 0.000, B 0.000, C 0.000 }
gfCNCPoint4[4005] = {X 298.3067, Y 11.4795, Z -5.5000, A 0.000, B 0.000, C 0.000 }
gfCNCPoint4[4006] = {X 298.4763, Y 10.4755, Z -5.5000, A 0.000, B 0.000, C 0.000 }
gfCNCPoint4[4007] = {X 298.7842, Y 9.5049, Z -5.5000, A 0.000, B 0.000, C 0.000 }
gfCNCPoint4[4008] = {X 298.7842, Y 7.1049, Z -5.5000, A 0.000, B 0.000, C 0.000 }
gfCNCPoint4[4009] = {X 233.3041, Y 7.1049, Z -5.5000, A 0.000, B 0.000, C 0.000 }
gfCNCPoint4[4010] = {X 233.3041, Y 11.9049, Z -5.5000, A 0.000, B 0.000, C 0.000 }
gfCNCPoint4[4011] = {X 233.1564, Y 11.9049, Z -5.5000, A 0.000, B 0.000, C 0.000 }
gfCNCPoint4[4012] = {X 233.1594, Y 12.0445, Z -5.5000, A 0.000, B 0.000, C 0.000 }
gfCNCPoint4[4013] = {X 233.1605, Y 12.1841, Z -5.5000, A 0.000, B 0.000, C 0.000 }
gfCNCPoint4[4014] = {X 233.2317, Y 12.0442, Z -5.5000, A 0.000, B 0.000, C 0.000 }
gfCNCPoint4[4015] = {X 233.3041, Y 11.9049, Z -5.5000, A 0.000, B 0.000, C 0.000 }
gfCNCPoint4[4016] = {X 233.3041, Y 9.5049, Z -5.5000, A 0.000, B 0.000, C 0.000 }
gfCNCPoint4[4017] = {X 230.2485, Y 9.5049, Z -5.5000, A 0.000, B 0.000, C 0.000 }
gfCNCPoint4[4018] = {X 230.6107, Y 10.7177, Z -5.5000, A 0.000, B 0.000, C 0.000 }
gfCNCPoint4[4019] = {X 230.7574, Y 11.9748, Z -5.5000, A 0.000, B 0.000, C 0.000 }
gfCNCPoint4[4020] = {X 230.7597, Y 12.0808, Z -5.5000, A 0.000, B 0.000, C 0.000 }
gfCNCPoint4[4021] = {X 230.7605, Y 12.1868, Z -5.5000, A 0.000, B 0.000, C 0.000 }
gfCNCPoint4[4022] = {X 230.7602, Y 13.0462, Z -5.5000, A 0.000, B 0.000, C 0.000 }
gfCNCPoint4[4023] = {X 230.6532, Y 14.2234, Z -5.5000, A 0.000, B 0.000, C 0.000 }
gfCNCPoint4[4024] = {X 230.3571, Y 15.3678, Z -5.5000, A 0.000, B 0.000, C 0.000 }
gfCNCPoint4[4025] = {X 229.8797, Y 16.4491, Z -5.5000, A 0.000, B 0.000, C 0.000 }
gfCNCPoint4[4026] = {X 229.2336, Y 17.4390, Z -5.5000, A 0.000, B 0.000, C 0.000 }
gfCNCPoint4[4027] = {X 229.2339, Y 25.8541, Z -5.5000, A 0.000, B 0.000, C 0.000 }
gfCNCPoint4[4028] = {X 231.6339, Y 25.8540, Z -5.5000, A 0.000, B 0.000, C 0.000 }
gfCNCPoint4[4029] = {X 231.6344, Y 38.9919, Z -5.5000, A 0.000, B 0.000, C 0.000 }
gfCNCPoint4[4030] = {X 231.6440, Y 39.0069, Z -5.5000, A 0.000, B 0.000, C 0.000 }
gfCNCPoint4[4031] = {X 232.3931, Y 37.9855, Z -5.5000, A 0.000, B 0.000, C 0.000 }
gfCNCPoint4[4032] = {X 233.2692, Y 37.0706, Z -5.5000, A 0.000, B 0.000, C 0.000 }
gfCNCPoint4[4033] = {X 234.2573, Y 36.2780, Z -5.5000, A 0.000, B 0.000, C 0.000 }
gfCNCPoint4[4034] = {X 235.5692, Y 33.7101, Z -5.5000, A 0.000, B 0.000, C 0.000 }
gfCNCPoint4[4035] = {X 234.4284, Y 32.2858, Z -5.5000, A 0.000, B 0.000, C 0.000 }
gfCNCPoint4[4036] = {X 233.4500, Y 30.7455, Z -5.5000, A 0.000, B 0.000, C 0.000 }
gfCNCPoint4[4037] = {X 232.6457, Y 29.1074, Z -5.5000, A 0.000, B 0.000, C 0.000 }
gfCNCPoint4[4038] = {X 232.0252, Y 27.3913, Z -5.5000, A 0.000, B 0.000, C 0.000 }
gfCNCPoint4[4039] = {X 231.8156, Y 26.6262, Z -5.5000, A 0.000, B 0.000, C 0.000 }
gfCNCPoint4[4040] = {X 231.6339, Y 25.8540, Z -5.5000, A 0.000, B 0.000, C 0.000 }
gfCNCPoint4[4041] = {X 229.2339, Y 25.8541, Z -5.5000, A 0.000, B 0.000, C 0.000 }
gfCNCPoint4[4042] = {X 229.2344, Y 39.7489, Z -5.5000, A 0.000, B 0.000, C 0.000 }
gfCNCPoint4[4043] = {X 229.4335, Y 40.0183, Z -5.5000, A 0.000, B 0.000, C 0.000 }
gfCNCPoint4[4044] = {X 229.6200, Y 40.2966, Z -5.5000, A 0.000, B 0.000, C 0.000 }
gfCNCPoint4[4045] = {X 230.1055, Y 41.1910, Z -5.5000, A 0.000, B 0.000, C 0.000 }
gfCNCPoint4[4046] = {X 230.4616, Y 42.1443, Z -5.5000, A 0.000, B 0.000, C 0.000 }
gfCNCPoint4[4047] = {X 230.6813, Y 43.1379, Z -5.5000, A 0.000, B 0.000, C 0.000 }
gfCNCPoint4[4048] = {X 230.7603, Y 44.1524, Z -5.5000, A 0.000, B 0.000, C 0.000 }
gfCNCPoint4[4049] = {X 230.7605, Y 45.0000, Z -5.5000, A 0.000, B 0.000, C 0.000 }
gfCNCPoint4[4050] = {X 230.7459, Y 45.4609, Z -5.5000, A 0.000, B 0.000, C 0.000 }
gfCNCPoint4[4051] = {X 230.7021, Y 45.9200, Z -5.5000, A 0.000, B 0.000, C 0.000 }
gfCNCPoint4[4052] = {X 232.5859, Y 45.9200, Z -5.5000, A 0.000, B 0.000, C 0.000 }
gfCNCPoint4[4053] = {X 232.5421, Y 45.4609, Z -5.5000, A 0.000, B 0.000, C 0.000 }
gfCNCPoint4[4054] = {X 232.5275, Y 45.0000, Z -5.5000, A 0.000, B 0.000, C 0.000 }
gfCNCPoint4[4055] = {X 232.5275, Y 44.2089, Z -5.5000, A 0.000, B 0.000, C 0.000 }
gfCNCPoint4[4056] = {X 232.6006, Y 43.1798, Z -5.5000, A 0.000, B 0.000, C 0.000 }
gfCNCPoint4[4057] = {X 232.8184, Y 42.1714, Z -5.5000, A 0.000, B 0.000, C 0.000 }
gfCNCPoint4[4058] = {X 233.1766, Y 41.2038, Z -5.5000, A 0.000, B 0.000, C 0.000 }
gfCNCPoint4[4059] = {X 233.6680, Y 40.2966, Z -5.5000, A 0.000, B 0.000, C 0.000 }
gfCNCPoint4[4060] = {X 234.3527, Y 39.3876, Z -5.5000, A 0.000, B 0.000, C 0.000 }
gfCNCPoint4[4061] = {X 235.1707, Y 38.5964, Z -5.5000, A 0.000, B 0.000, C 0.000 }
gfCNCPoint4[4062] = {X 236.1021, Y 37.9424, Z -5.5000, A 0.000, B 0.000, C 0.000 }
gfCNCPoint4[4063] = {X 238.4998, Y 33.2491, Z -5.5000, A 0.000, B 0.000, C 0.000 }
gfCNCPoint4[4064] = {X 237.3860, Y 32.1412, Z -5.5000, A 0.000, B 0.000, C 0.000 }
gfCNCPoint4[4065] = {X 236.4006, Y 30.9178, Z -5.5000, A 0.000, B 0.000, C 0.000 }
gfCNCPoint4[4066] = {X 235.5556, Y 29.5935, Z -5.5000, A 0.000, B 0.000, C 0.000 }
gfCNCPoint4[4067] = {X 234.8612, Y 28.1844, Z -5.5000, A 0.000, B 0.000, C 0.000 }
gfCNCPoint4[4068] = {X 234.3257, Y 26.7075, Z -5.5000, A 0.000, B 0.000, C 0.000 }
gfCNCPoint4[4069] = {X 234.1404, Y 26.0302, Z -5.5000, A 0.000, B 0.000, C 0.000 }
gfCNCPoint4[4070] = {X 233.9797, Y 25.3467, Z -5.5000, A 0.000, B 0.000, C 0.000 }
gfCNCPoint4[4071] = {X 233.6673, Y 23.4576, Z -5.5000, A 0.000, B 0.000, C 0.000 }
gfCNCPoint4[4072] = {X 233.5417, Y 21.5470, Z -5.5000, A 0.000, B 0.000, C 0.000 }
gfCNCPoint4[4073] = {X 233.6042, Y 19.6333, Z -5.5000, A 0.000, B 0.000, C 0.000 }
gfCNCPoint4[4074] = {X 233.8541, Y 17.7350, Z -5.5000, A 0.000, B 0.000, C 0.000 }
gfCNCPoint4[4075] = {X 234.2890, Y 15.8703, Z -5.5000, A 0.000, B 0.000, C 0.000 }
gfCNCPoint4[4076] = {X 234.7351, Y 14.5423, Z -5.5000, A 0.000, B 0.000, C 0.000 }
gfCNCPoint4[4077] = {X 235.3046, Y 13.2625, Z -5.5000, A 0.000, B 0.000, C 0.000 }
gfCNCPoint4[4078] = {X 235.3658, Y 13.1421, Z -5.5000, A 0.000, B 0.000, C 0.000 }
gfCNCPoint4[4079] = {X 235.4282, Y 13.0222, Z -5.5000, A 0.000, B 0.000, C 0.000 }
gfCNCPoint4[4080] = {X 236.1695, Y 11.7670, Z -5.5000, A 0.000, B 0.000, C 0.000 }
gfCNCPoint4[4081] = {X 237.0306, Y 10.5908, Z -5.5000, A 0.000, B 0.000, C 0.000 }
gfCNCPoint4[4082] = {X 238.0032, Y 9.5049, Z -5.5000, A 0.000, B 0.000, C 0.000 }
gfCNCPoint4[4083] = {X 233.3041, Y 9.5049, Z -5.5000, A 0.000, B 0.000, C 0.000 }
gfCNCPoint4[4084] = {X 233.3041, Y 7.1049, Z -5.5000, A 0.000, B 0.000, C 0.000 }
gfCNCPoint4[4085] = {X 191.0937, Y 7.1049, Z -5.5000, A 0.000, B 0.000, C 0.000 }
gfCNCPoint4[4086] = {X 193.0670, Y 7.6381, Z -5.5000, A 0.000, B 0.000, C 0.000 }
gfCNCPoint4[4087] = {X 194.9657, Y 8.3955, Z -5.5000, A 0.000, B 0.000, C 0.000 }
gfCNCPoint4[4088] = {X 196.7641, Y 9.3671, Z -5.5000, A 0.000, B 0.000, C 0.000 }
gfCNCPoint4[4089] = {X 198.4384, Y 10.5398, Z -5.5000, A 0.000, B 0.000, C 0.000 }
gfCNCPoint4[4090] = {X 198.8599, Y 10.8895, Z -5.5000, A 0.000, B 0.000, C 0.000 }
gfCNCPoint4[4091] = {X 199.2669, Y 11.2560, Z -5.5000, A 0.000, B 0.000, C 0.000 }
gfCNCPoint4[4092] = {X 200.3520, Y 12.3983, Z -5.5000, A 0.000, B 0.000, C 0.000 }
gfCNCPoint4[4093] = {X 201.2976, Y 13.6587, Z -5.5000, A 0.000, B 0.000, C 0.000 }
gfCNCPoint4[4094] = {X 202.0908, Y 15.0201, Z -5.5000, A 0.000, B 0.000, C 0.000 }
gfCNCPoint4[4095] = {X 202.7210, Y 16.4641, Z -5.5000, A 0.000, B 0.000, C 0.000 }
gfCNCPoint4[4096] = {X 203.2147, Y 18.1838, Z -5.5000, A 0.000, B 0.000, C 0.000 }
gfCNCPoint4[4097] = {X 203.5079, Y 19.9487, Z -5.5000, A 0.000, B 0.000, C 0.000 }
gfCNCPoint4[4098] = {X 203.5970, Y 21.7356, Z -5.5000, A 0.000, B 0.000, C 0.000 }
gfCNCPoint4[4099] = {X 203.4807, Y 23.5210, Z -5.5000, A 0.000, B 0.000, C 0.000 }
gfCNCPoint4[4100] = {X 203.1604, Y 25.2812, Z -5.5000, A 0.000, B 0.000, C 0.000 }
gfCNCPoint4[4101] = {X 202.7600, Y 26.6266, Z -5.5000, A 0.000, B 0.000, C 0.000 }
gfCNCPoint4[4102] = {X 202.2084, Y 27.9174, Z -5.5000, A 0.000, B 0.000, C 0.000 }
gfCNCPoint4[4103] = {X 201.5127, Y 29.1366, Z -5.5000, A 0.000, B 0.000, C 0.000 }
gfCNCPoint4[4104] = {X 200.6822, Y 30.2683, Z -5.5000, A 0.000, B 0.000, C 0.000 }
gfCNCPoint4[4105] = {X 199.7277, Y 31.2976, Z -5.5000, A 0.000, B 0.000, C 0.000 }
gfCNCPoint4[4106] = {X 200.5670, Y 31.8700, Z -5.5000, A 0.000, B 0.000, C 0.000 }
gfCNCPoint4[4107] = {X 201.2696, Y 32.6039, Z -5.5000, A 0.000, B 0.000, C 0.000 }
gfCNCPoint4[4108] = {X 201.8050, Y 33.4673, Z -5.5000, A 0.000, B 0.000, C 0.000 }
gfCNCPoint4[4109] = {X 204.8262, Y 39.7091, Z -5.5000, A 0.000, B 0.000, C 0.000 }
gfCNCPoint4[4110] = {X 205.1508, Y 40.5847, Z -5.5000, A 0.000, B 0.000, C 0.000 }
gfCNCPoint4[4111] = {X 205.3026, Y 41.5062, Z -5.5000, A 0.000, B 0.000, C 0.000 }
gfCNCPoint4[4112] = {X 205.2761, Y 42.4397, Z -5.5000, A 0.000, B 0.000, C 0.000 }
gfCNCPoint4[4113] = {X 205.0723, Y 43.3511, Z -5.5000, A 0.000, B 0.000, C 0.000 }
gfCNCPoint4[4114] = {X 204.6986, Y 44.2070, Z -5.5000, A 0.000, B 0.000, C 0.000 }
gfCNCPoint4[4115] = {X 204.1687, Y 44.9760, Z -5.5000, A 0.000, B 0.000, C 0.000 }
gfCNCPoint4[4116] = {X 203.5020, Y 45.6299, Z -5.5000, A 0.000, B 0.000, C 0.000 }
gfCNCPoint4[4117] = {X 202.9658, Y 46.0634, Z -5.5000, A 0.000, B 0.000, C 0.000 }
gfCNCPoint4[4118] = {X 202.2139, Y 46.5641, Z -5.5000, A 0.000, B 0.000, C 0.000 }
gfCNCPoint4[4119] = {X 201.3828, Y 46.9179, Z -5.5000, A 0.000, B 0.000, C 0.000 }
gfCNCPoint4[4120] = {X 200.5007, Y 47.1129, Z -5.5000, A 0.000, B 0.000, C 0.000 }
gfCNCPoint4[4121] = {X 199.5979, Y 47.1424, Z -5.5000, A 0.000, B 0.000, C 0.000 }
gfCNCPoint4[4122] = {X 198.7050, Y 47.0053, Z -5.5000, A 0.000, B 0.000, C 0.000 }
gfCNCPoint4[4123] = {X 197.7383, Y 47.5279, Z -5.5000, A 0.000, B 0.000, C 0.000 }
gfCNCPoint4[4124] = {X 196.7525, Y 48.0135, Z -5.5000, A 0.000, B 0.000, C 0.000 }
gfCNCPoint4[4125] = {X 199.8110, Y 54.5316, Z -5.5000, A 0.000, B 0.000, C 0.000 }
gfCNCPoint4[4126] = {X 197.5976, Y 55.4816, Z -5.5000, A 0.000, B 0.000, C 0.000 }
gfCNCPoint4[4127] = {X 195.3259, Y 56.2822, Z -5.5000, A 0.000, B 0.000, C 0.000 }
gfCNCPoint4[4128] = {X 195.3577, Y 56.6288, Z -5.5000, A 0.000, B 0.000, C 0.000 }
gfCNCPoint4[4129] = {X 195.3824, Y 56.9759, Z -5.5000, A 0.000, B 0.000, C 0.000 }
gfCNCPoint4[4130] = {X 199.6720, Y 61.6578, Z -5.5000, A 0.000, B 0.000, C 0.000 }
gfCNCPoint4[4131] = {X 199.5095, Y 60.3400, Z -5.5000, A 0.000, B 0.000, C 0.000 }
gfCNCPoint4[4132] = {X 199.4510, Y 59.0136, Z -5.5000, A 0.000, B 0.000, C 0.000 }
gfCNCPoint4[4133] = {X 199.4508, Y 58.0000, Z -5.5000, A 0.000, B 0.000, C 0.000 }
gfCNCPoint4[4134] = {X 199.5411, Y 56.2565, Z -5.5000, A 0.000, B 0.000, C 0.000 }
gfCNCPoint4[4135] = {X 199.8110, Y 54.5316, Z -5.5000, A 0.000, B 0.000, C 0.000 }
gfCNCPoint4[4136] = {X 198.7915, Y 52.3589, Z -5.5000, A 0.000, B 0.000, C 0.000 }
gfCNCPoint4[4137] = {X 196.1934, Y 53.4482, Z -5.5000, A 0.000, B 0.000, C 0.000 }
gfCNCPoint4[4138] = {X 193.5136, Y 54.3172, Z -5.5000, A 0.000, B 0.000, C 0.000 }
gfCNCPoint4[4139] = {X 193.0574, Y 54.4430, Z -5.5000, A 0.000, B 0.000, C 0.000 }
gfCNCPoint4[4140] = {X 192.5992, Y 54.5610, Z -5.5000, A 0.000, B 0.000, C 0.000 }
gfCNCPoint4[4141] = {X 192.9061, Y 56.2398, Z -5.5000, A 0.000, B 0.000, C 0.000 }
gfCNCPoint4[4142] = {X 193.0134, Y 57.9430, Z -5.5000, A 0.000, B 0.000, C 0.000 }
gfCNCPoint4[4143] = {X 210.3939, Y 76.9129, Z -5.5000, A 0.000, B 0.000, C 0.000 }
gfCNCPoint4[4144] = {X 212.1635, Y 75.2916, Z -5.5000, A 0.000, B 0.000, C 0.000 }
gfCNCPoint4[4145] = {X 215.1986, Y 78.6042, Z -5.5000, A 0.000, B 0.000, C 0.000 }
gfCNCPoint4[4146] = {X 218.3269, Y 76.6001, Z -5.5000, A 0.000, B 0.000, C 0.000 }
gfCNCPoint4[4147] = {X 216.9974, Y 76.0784, Z -5.5000, A 0.000, B 0.000, C 0.000 }
gfCNCPoint4[4148] = {X 216.3752, Y 75.8853, Z -5.5000, A 0.000, B 0.000, C 0.000 }
gfCNCPoint4[4149] = {X 215.7288, Y 75.8033, Z -5.5000, A 0.000, B 0.000, C 0.000 }
gfCNCPoint4[4150] = {X 213.9325, Y 75.6428, Z -5.5000, A 0.000, B 0.000, C 0.000 }
gfCNCPoint4[4151] = {X 212.1635, Y 75.2916, Z -5.5000, A 0.000, B 0.000, C 0.000 }
gfCNCPoint4[4152] = {X 210.3939, Y 76.9129, Z -5.5000, A 0.000, B 0.000, C 0.000 }
gfCNCPoint4[4153] = {X 214.7930, Y 81.7142, Z -5.5000, A 0.000, B 0.000, C 0.000 }
gfCNCPoint4[4154] = {X 223.5816, Y 76.0840, Z -5.5000, A 0.000, B 0.000, C 0.000 }
gfCNCPoint4[4155] = {X 217.8863, Y 73.8490, Z -5.5000, A 0.000, B 0.000, C 0.000 }
gfCNCPoint4[4156] = {X 216.8712, Y 73.5371, Z -5.5000, A 0.000, B 0.000, C 0.000 }
gfCNCPoint4[4157] = {X 215.8174, Y 73.4050, Z -5.5000, A 0.000, B 0.000, C 0.000 }
gfCNCPoint4[4158] = {X 214.2750, Y 73.2674, Z -5.5000, A 0.000, B 0.000, C 0.000 }
gfCNCPoint4[4159] = {X 212.7560, Y 72.9659, Z -5.5000, A 0.000, B 0.000, C 0.000 }
gfCNCPoint4[4160] = {X 211.1570, Y 72.4582, Z -5.5000, A 0.000, B 0.000, C 0.000 }
gfCNCPoint4[4161] = {X 209.6274, Y 71.7690, Z -5.5000, A 0.000, B 0.000, C 0.000 }
gfCNCPoint4[4162] = {X 208.1878, Y 70.9075, Z -5.5000, A 0.000, B 0.000, C 0.000 }
gfCNCPoint4[4163] = {X 206.8575, Y 69.8852, Z -5.5000, A 0.000, B 0.000, C 0.000 }
gfCNCPoint4[4164] = {X 205.6544, Y 68.7159, Z -5.5000, A 0.000, B 0.000, C 0.000 }
gfCNCPoint4[4165] = {X 204.5946, Y 67.4154, Z -5.5000, A 0.000, B 0.000, C 0.000 }
gfCNCPoint4[4166] = {X 203.6924, Y 66.0010, Z -5.5000, A 0.000, B 0.000, C 0.000 }
gfCNCPoint4[4167] = {X 202.9598, Y 64.4917, Z -5.5000, A 0.000, B 0.000, C 0.000 }
gfCNCPoint4[4168] = {X 202.4067, Y 62.9078, Z -5.5000, A 0.000, B 0.000, C 0.000 }
gfCNCPoint4[4169] = {X 202.0405, Y 61.2705, Z -5.5000, A 0.000, B 0.000, C 0.000 }
gfCNCPoint4[4170] = {X 201.9013, Y 60.1426, Z -5.5000, A 0.000, B 0.000, C 0.000 }
gfCNCPoint4[4171] = {X 201.8510, Y 59.0073, Z -5.5000, A 0.000, B 0.000, C 0.000 }
gfCNCPoint4[4172] = {X 201.8508, Y 58.0000, Z -5.5000, A 0.000, B 0.000, C 0.000 }
gfCNCPoint4[4173] = {X 201.9283, Y 56.5044, Z -5.5000, A 0.000, B 0.000, C 0.000 }
gfCNCPoint4[4174] = {X 202.1598, Y 55.0248, Z -5.5000, A 0.000, B 0.000, C 0.000 }
gfCNCPoint4[4175] = {X 202.4965, Y 53.7243, Z -5.5000, A 0.000, B 0.000, C 0.000 }
gfCNCPoint4[4176] = {X 202.9523, Y 52.4606, Z -5.5000, A 0.000, B 0.000, C 0.000 }
gfCNCPoint4[4177] = {X 203.5232, Y 51.2445, Z -5.5000, A 0.000, B 0.000, C 0.000 }
gfCNCPoint4[4178] = {X 202.2640, Y 51.6560, Z -5.5000, A 0.000, B 0.000, C 0.000 }
gfCNCPoint4[4179] = {X 200.9604, Y 51.8919, Z -5.5000, A 0.000, B 0.000, C 0.000 }
gfCNCPoint4[4180] = {X 199.6369, Y 51.9478, Z -5.5000, A 0.000, B 0.000, C 0.000 }
gfCNCPoint4[4181] = {X 199.2156, Y 52.1563, Z -5.5000, A 0.000, B 0.000, C 0.000 }
gfCNCPoint4[4182] = {X 198.7915, Y 52.3589, Z -5.5000, A 0.000, B 0.000, C 0.000 }
gfCNCPoint4[4183] = {X 197.7720, Y 50.1862, Z -5.5000, A 0.000, B 0.000, C 0.000 }
gfCNCPoint4[4184] = {X 195.3553, Y 51.1993, Z -5.5000, A 0.000, B 0.000, C 0.000 }
gfCNCPoint4[4185] = {X 192.8625, Y 52.0072, Z -5.5000, A 0.000, B 0.000, C 0.000 }
gfCNCPoint4[4186] = {X 192.4424, Y 52.1231, Z -5.5000, A 0.000, B 0.000, C 0.000 }
gfCNCPoint4[4187] = {X 192.0205, Y 52.2318, Z -5.5000, A 0.000, B 0.000, C 0.000 }
gfCNCPoint4[4188] = {X 190.7203, Y 52.5188, Z -5.5000, A 0.000, B 0.000, C 0.000 }
gfCNCPoint4[4189] = {X 189.4069, Y 52.7373, Z -5.5000, A 0.000, B 0.000, C 0.000 }
gfCNCPoint4[4190] = {X 189.9005, Y 53.9114, Z -5.5000, A 0.000, B 0.000, C 0.000 }
gfCNCPoint4[4191] = {X 190.2679, Y 55.1310, Z -5.5000, A 0.000, B 0.000, C 0.000 }
gfCNCPoint4[4192] = {X 190.5268, Y 56.5551, Z -5.5000, A 0.000, B 0.000, C 0.000 }
gfCNCPoint4[4193] = {X 190.6135, Y 58.0000, Z -5.5000, A 0.000, B 0.000, C 0.000 }
gfCNCPoint4[4194] = {X 190.6132, Y 58.8760, Z -5.5000, A 0.000, B 0.000, C 0.000 }
gfCNCPoint4[4195] = {X 214.3875, Y 84.8243, Z -5.5000, A 0.000, B 0.000, C 0.000 }
gfCNCPoint4[4196] = {X 228.8363, Y 75.5679, Z -5.5000, A 0.000, B 0.000, C 0.000 }
gfCNCPoint4[4197] = {X 218.7733, Y 71.6189, Z -5.5000, A 0.000, B 0.000, C 0.000 }
gfCNCPoint4[4198] = {X 217.8429, Y 71.3049, Z -5.5000, A 0.000, B 0.000, C 0.000 }
gfCNCPoint4[4199] = {X 216.8827, Y 71.0999, Z -5.5000, A 0.000, B 0.000, C 0.000 }
gfCNCPoint4[4200] = {X 215.9052, Y 71.0066, Z -5.5000, A 0.000, B 0.000, C 0.000 }
gfCNCPoint4[4201] = {X 214.2355, Y 70.8310, Z -5.5000, A 0.000, B 0.000, C 0.000 }
gfCNCPoint4[4202] = {X 212.6062, Y 70.4255, Z -5.5000, A 0.000, B 0.000, C 0.000 }
gfCNCPoint4[4203] = {X 211.0489, Y 69.7981, Z -5.5000, A 0.000, B 0.000, C 0.000 }
gfCNCPoint4[4204] = {X 209.5937, Y 68.9609, Z -5.5000, A 0.000, B 0.000, C 0.000 }
gfCNCPoint4[4205] = {X 208.2685, Y 67.9300, Z -5.5000, A 0.000, B 0.000, C 0.000 }
gfCNCPoint4[4206] = {X 207.0991, Y 66.7253, Z -5.5000, A 0.000, B 0.000, C 0.000 }
gfCNCPoint4[4207] = {X 206.1081, Y 65.3701, Z -5.5000, A 0.000, B 0.000, C 0.000 }
gfCNCPoint4[4208] = {X 205.3145, Y 63.8905, Z -5.5000, A 0.000, B 0.000, C 0.000 }
gfCNCPoint4[4209] = {X 204.7337, Y 62.3153, Z -5.5000, A 0.000, B 0.000, C 0.000 }
gfCNCPoint4[4210] = {X 204.3769, Y 60.6747, Z -5.5000, A 0.000, B 0.000, C 0.000 }
gfCNCPoint4[4211] = {X 204.2510, Y 59.0005, Z -5.5000, A 0.000, B 0.000, C 0.000 }
gfCNCPoint4[4212] = {X 204.2508, Y 58.0000, Z -5.5000, A 0.000, B 0.000, C 0.000 }
gfCNCPoint4[4213] = {X 204.3396, Y 56.5378, Z -5.5000, A 0.000, B 0.000, C 0.000 }
gfCNCPoint4[4214] = {X 204.6048, Y 55.0970, Z -5.5000, A 0.000, B 0.000, C 0.000 }
gfCNCPoint4[4215] = {X 205.0424, Y 53.6990, Z -5.5000, A 0.000, B 0.000, C 0.000 }
gfCNCPoint4[4216] = {X 205.6460, Y 52.3642, Z -5.5000, A 0.000, B 0.000, C 0.000 }
gfCNCPoint4[4217] = {X 206.5296, Y 50.9387, Z -5.5000, A 0.000, B 0.000, C 0.000 }
gfCNCPoint4[4218] = {X 207.6020, Y 49.6493, Z -5.5000, A 0.000, B 0.000, C 0.000 }
gfCNCPoint4[4219] = {X 208.8427, Y 48.5209, Z -5.5000, A 0.000, B 0.000, C 0.000 }
gfCNCPoint4[4220] = {X 210.2277, Y 47.5751, Z -5.5000, A 0.000, B 0.000, C 0.000 }
gfCNCPoint4[4221] = {X 209.8801, Y 46.3328, Z -5.5000, A 0.000, B 0.000, C 0.000 }
gfCNCPoint4[4222] = {X 209.7572, Y 45.0487, Z -5.5000, A 0.000, B 0.000, C 0.000 }
gfCNCPoint4[4223] = {X 209.7570, Y 44.1949, Z -5.5000, A 0.000, B 0.000, C 0.000 }
gfCNCPoint4[4224] = {X 209.8558, Y 43.0053, Z -5.5000, A 0.000, B 0.000, C 0.000 }
gfCNCPoint4[4225] = {X 210.1496, Y 41.8484, Z -5.5000, A 0.000, B 0.000, C 0.000 }
gfCNCPoint4[4226] = {X 210.6302, Y 40.7557, Z -5.5000, A 0.000, B 0.000, C 0.000 }
gfCNCPoint4[4227] = {X 211.2845, Y 39.7574, Z -5.5000, A 0.000, B 0.000, C 0.000 }
gfCNCPoint4[4228] = {X 211.2845, Y 37.0761, Z -5.5000, A 0.000, B 0.000, C 0.000 }
gfCNCPoint4[4229] = {X 208.8845, Y 37.0761, Z -5.5000, A 0.000, B 0.000, C 0.000 }
gfCNCPoint4[4230] = {X 208.8845, Y 18.1972, Z -5.5000, A 0.000, B 0.000, C 0.000 }
gfCNCPoint4[4231] = {X 208.2327, Y 17.0013, Z -5.5000, A 0.000, B 0.000, C 0.000 }
gfCNCPoint4[4232] = {X 207.7552, Y 15.7257, Z -5.5000, A 0.000, B 0.000, C 0.000 }
gfCNCPoint4[4233] = {X 207.4614, Y 14.3958, Z -5.5000, A 0.000, B 0.000, C 0.000 }
gfCNCPoint4[4234] = {X 207.3572, Y 13.0378, Z -5.5000, A 0.000, B 0.000, C 0.000 }
gfCNCPoint4[4235] = {X 207.3570, Y 12.1868, Z -5.5000, A 0.000, B 0.000, C 0.000 }
gfCNCPoint4[4236] = {X 207.3580, Y 12.0459, Z -5.5000, A 0.000, B 0.000, C 0.000 }
gfCNCPoint4[4237] = {X 207.3611, Y 11.9049, Z -5.5000, A 0.000, B 0.000, C 0.000 }
gfCNCPoint4[4238] = {X 205.8575, Y 11.9049, Z -5.5000, A 0.000, B 0.000, C 0.000 }
gfCNCPoint4[4239] = {X 206.6126, Y 13.3419, Z -5.5000, A 0.000, B 0.000, C 0.000 }
gfCNCPoint4[4240] = {X 207.2380, Y 14.8398, Z -5.5000, A 0.000, B 0.000, C 0.000 }
gfCNCPoint4[4241] = {X 207.7988, Y 16.7126, Z -5.5000, A 0.000, B 0.000, C 0.000 }
gfCNCPoint4[4242] = {X 208.1776, Y 18.6305, Z -5.5000, A 0.000, B 0.000, C 0.000 }
gfCNCPoint4[4243] = {X 208.3709, Y 20.5759, Z -5.5000, A 0.000, B 0.000, C 0.000 }
gfCNCPoint4[4244] = {X 208.3770, Y 22.5308, Z -5.5000, A 0.000, B 0.000, C 0.000 }
gfCNCPoint4[4245] = {X 208.1957, Y 24.4773, Z -5.5000, A 0.000, B 0.000, C 0.000 }
gfCNCPoint4[4246] = {X 207.8288, Y 26.3975, Z -5.5000, A 0.000, B 0.000, C 0.000 }
gfCNCPoint4[4247] = {X 207.3617, Y 28.0100, Z -5.5000, A 0.000, B 0.000, C 0.000 }
gfCNCPoint4[4248] = {X 206.7383, Y 29.5688, Z -5.5000, A 0.000, B 0.000, C 0.000 }
gfCNCPoint4[4249] = {X 205.9646, Y 31.0587, Z -5.5000, A 0.000, B 0.000, C 0.000 }
gfCNCPoint4[4250] = {X 206.0465, Y 31.2166, Z -5.5000, A 0.000, B 0.000, C 0.000 }
gfCNCPoint4[4251] = {X 206.1255, Y 31.3761, Z -5.5000, A 0.000, B 0.000, C 0.000 }
gfCNCPoint4[4252] = {X 208.8845, Y 37.0761, Z -5.5000, A 0.000, B 0.000, C 0.000 }
gfCNCPoint4[4253] = {X 211.2845, Y 37.0761, Z -5.5000, A 0.000, B 0.000, C 0.000 }
gfCNCPoint4[4254] = {X 211.2843, Y 17.4394, Z -5.5000, A 0.000, B 0.000, C 0.000 }
gfCNCPoint4[4255] = {X 210.6360, Y 16.4458, Z -5.5000, A 0.000, B 0.000, C 0.000 }
gfCNCPoint4[4256] = {X 210.1577, Y 15.3600, Z -5.5000, A 0.000, B 0.000, C 0.000 }
gfCNCPoint4[4257] = {X 209.8622, Y 14.2109, Z -5.5000, A 0.000, B 0.000, C 0.000 }
gfCNCPoint4[4258] = {X 209.7572, Y 13.0291, Z -5.5000, A 0.000, B 0.000, C 0.000 }
gfCNCPoint4[4259] = {X 209.7570, Y 12.1868, Z -5.5000, A 0.000, B 0.000, C 0.000 }
gfCNCPoint4[4260] = {X 209.7578, Y 12.0808, Z -5.5000, A 0.000, B 0.000, C 0.000 }
gfCNCPoint4[4261] = {X 209.7601, Y 11.9748, Z -5.5000, A 0.000, B 0.000, C 0.000 }
gfCNCPoint4[4262] = {X 209.9068, Y 10.7177, Z -5.5000, A 0.000, B 0.000, C 0.000 }
gfCNCPoint4[4263] = {X 210.2690, Y 9.5049, Z -5.5000, A 0.000, B 0.000, C 0.000 }
gfCNCPoint4[4264] = {X 200.9082, Y 9.5049, Z -5.5000, A 0.000, B 0.000, C 0.000 }
gfCNCPoint4[4265] = {X 201.9818, Y 10.6134, Z -5.5000, A 0.000, B 0.000, C 0.000 }
gfCNCPoint4[4266] = {X 202.9435, Y 11.8201, Z -5.5000, A 0.000, B 0.000, C 0.000 }
gfCNCPoint4[4267] = {X 203.7844, Y 13.1140, Z -5.5000, A 0.000, B 0.000, C 0.000 }
gfCNCPoint4[4268] = {X 204.4377, Y 14.3567, Z -5.5000, A 0.000, B 0.000, C 0.000 }
gfCNCPoint4[4269] = {X 204.9795, Y 15.6519, Z -5.5000, A 0.000, B 0.000, C 0.000 }
gfCNCPoint4[4270] = {X 205.5519, Y 17.6384, Z -5.5000, A 0.000, B 0.000, C 0.000 }
gfCNCPoint4[4271] = {X 205.8926, Y 19.6775, Z -5.5000, A 0.000, B 0.000, C 0.000 }
gfCNCPoint4[4272] = {X 205.9970, Y 21.7422, Z -5.5000, A 0.000, B 0.000, C 0.000 }
gfCNCPoint4[4273] = {X 205.8638, Y 23.8052, Z -5.5000, A 0.000, B 0.000, C 0.000 }
gfCNCPoint4[4274] = {X 205.4947, Y 25.8393, Z -5.5000, A 0.000, B 0.000, C 0.000 }
gfCNCPoint4[4275] = {X 205.0935, Y 27.2256, Z -5.5000, A 0.000, B 0.000, C 0.000 }
gfCNCPoint4[4276] = {X 204.5579, Y 28.5658, Z -5.5000, A 0.000, B 0.000, C 0.000 }
gfCNCPoint4[4277] = {X 203.8931, Y 29.8467, Z -5.5000, A 0.000, B 0.000, C 0.000 }
gfCNCPoint4[4278] = {X 203.1056, Y 31.0561, Z -5.5000, A 0.000, B 0.000, C 0.000 }
gfCNCPoint4[4279] = {X 203.5734, Y 31.7150, Z -5.5000, A 0.000, B 0.000, C 0.000 }
gfCNCPoint4[4280] = {X 203.9653, Y 32.4217, Z -5.5000, A 0.000, B 0.000, C 0.000 }
gfCNCPoint4[4281] = {X 206.9865, Y 38.6634, Z -5.5000, A 0.000, B 0.000, C 0.000 }
gfCNCPoint4[4282] = {X 207.4240, Y 39.8017, Z -5.5000, A 0.000, B 0.000, C 0.000 }
gfCNCPoint4[4283] = {X 207.6653, Y 40.9971, Z -5.5000, A 0.000, B 0.000, C 0.000 }
gfCNCPoint4[4284] = {X 207.7038, Y 42.2159, Z -5.5000, A 0.000, B 0.000, C 0.000 }
gfCNCPoint4[4285] = {X 207.5382, Y 43.4241, Z -5.5000, A 0.000, B 0.000, C 0.000 }
gfCNCPoint4[4286] = {X 207.1733, Y 44.5877, Z -5.5000, A 0.000, B 0.000, C 0.000 }
gfCNCPoint4[4287] = {X 206.6193, Y 45.6741, Z -5.5000, A 0.000, B 0.000, C 0.000 }
gfCNCPoint4[4288] = {X 205.8917, Y 46.6527, Z -5.5000, A 0.000, B 0.000, C 0.000 }
gfCNCPoint4[4289] = {X 205.0110, Y 47.4962, Z -5.5000, A 0.000, B 0.000, C 0.000 }
gfCNCPoint4[4290] = {X 204.4748, Y 47.9297, Z -5.5000, A 0.000, B 0.000, C 0.000 }
gfCNCPoint4[4291] = {X 203.5895, Y 48.5432, Z -5.5000, A 0.000, B 0.000, C 0.000 }
gfCNCPoint4[4292] = {X 202.6236, Y 49.0195, Z -5.5000, A 0.000, B 0.000, C 0.000 }
gfCNCPoint4[4293] = {X 201.4896, Y 49.3736, Z -5.5000, A 0.000, B 0.000, C 0.000 }
gfCNCPoint4[4294] = {X 200.3131, Y 49.5389, Z -5.5000, A 0.000, B 0.000, C 0.000 }
gfCNCPoint4[4295] = {X 199.1254, Y 49.5109, Z -5.5000, A 0.000, B 0.000, C 0.000 }
gfCNCPoint4[4296] = {X 198.4528, Y 49.8567, Z -5.5000, A 0.000, B 0.000, C 0.000 }
gfCNCPoint4[4297] = {X 197.7720, Y 50.1862, Z -5.5000, A 0.000, B 0.000, C 0.000 }
gfCNCPoint4[4298] = {X 196.7525, Y 48.0135, Z -5.5000, A 0.000, B 0.000, C 0.000 }
gfCNCPoint4[4299] = {X 194.5171, Y 48.9504, Z -5.5000, A 0.000, B 0.000, C 0.000 }
gfCNCPoint4[4300] = {X 192.2113, Y 49.6972, Z -5.5000, A 0.000, B 0.000, C 0.000 }
gfCNCPoint4[4301] = {X 190.6549, Y 50.0835, Z -5.5000, A 0.000, B 0.000, C 0.000 }
gfCNCPoint4[4302] = {X 189.0754, Y 50.3603, Z -5.5000, A 0.000, B 0.000, C 0.000 }
gfCNCPoint4[4303] = {X 186.8990, Y 50.5588, Z -5.5000, A 0.000, B 0.000, C 0.000 }
gfCNCPoint4[4304] = {X 184.7136, Y 50.5496, Z -5.5000, A 0.000, B 0.000, C 0.000 }
gfCNCPoint4[4305] = {X 184.7384, Y 50.0702, Z -5.5000, A 0.000, B 0.000, C 0.000 }
gfCNCPoint4[4306] = {X 182.7584, Y 49.8795, Z -5.5000, A 0.000, B 0.000, C 0.000 }
gfCNCPoint4[4307] = {X 180.8029, Y 49.5145, Z -5.5000, A 0.000, B 0.000, C 0.000 }
gfCNCPoint4[4308] = {X 178.9541, Y 48.9786, Z -5.5000, A 0.000, B 0.000, C 0.000 }
gfCNCPoint4[4309] = {X 177.1795, Y 48.2332, Z -5.5000, A 0.000, B 0.000, C 0.000 }
gfCNCPoint4[4310] = {X 175.5025, Y 47.2882, Z -5.5000, A 0.000, B 0.000, C 0.000 }
gfCNCPoint4[4311] = {X 173.9457, Y 46.1563, Z -5.5000, A 0.000, B 0.000, C 0.000 }
gfCNCPoint4[4312] = {X 172.7973, Y 45.1084, Z -5.5000, A 0.000, B 0.000, C 0.000 }
gfCNCPoint4[4313] = {X 171.7812, Y 43.9320, Z -5.5000, A 0.000, B 0.000, C 0.000 }
gfCNCPoint4[4314] = {X 170.9114, Y 42.6436, Z -5.5000, A 0.000, B 0.000, C 0.000 }
gfCNCPoint4[4315] = {X 170.2004, Y 41.2612, Z -5.5000, A 0.000, B 0.000, C 0.000 }
gfCNCPoint4[4316] = {X 169.6580, Y 39.8043, Z -5.5000, A 0.000, B 0.000, C 0.000 }
gfCNCPoint4[4317] = {X 169.2919, Y 38.2935, Z -5.5000, A 0.000, B 0.000, C 0.000 }
gfCNCPoint4[4318] = {X 169.1814, Y 37.5992, Z -5.5000, A 0.000, B 0.000, C 0.000 }
gfCNCPoint4[4319] = {X 169.0222, Y 35.9860, Z -5.5000, A 0.000, B 0.000, C 0.000 }
gfCNCPoint4[4320] = {X 169.0393, Y 34.3651, Z -5.5000, A 0.000, B 0.000, C 0.000 }
gfCNCPoint4[4321] = {X 169.2324, Y 32.7556, Z -5.5000, A 0.000, B 0.000, C 0.000 }
gfCNCPoint4[4322] = {X 169.5992, Y 31.1767, Z -5.5000, A 0.000, B 0.000, C 0.000 }
gfCNCPoint4[4323] = {X 170.1355, Y 29.6469, Z -5.5000, A 0.000, B 0.000, C 0.000 }
gfCNCPoint4[4324] = {X 170.7624, Y 28.3592, Z -5.5000, A 0.000, B 0.000, C 0.000 }
gfCNCPoint4[4325] = {X 171.5522, Y 27.1645, Z -5.5000, A 0.000, B 0.000, C 0.000 }
gfCNCPoint4[4326] = {X 172.4913, Y 26.0832, Z -5.5000, A 0.000, B 0.000, C 0.000 }
gfCNCPoint4[4327] = {X 173.5637, Y 25.1340, Z -5.5000, A 0.000, B 0.000, C 0.000 }
gfCNCPoint4[4328] = {X 174.7509, Y 24.3329, Z -5.5000, A 0.000, B 0.000, C 0.000 }
gfCNCPoint4[4329] = {X 173.9909, Y 23.9226, Z -5.5000, A 0.000, B 0.000, C 0.000 }
gfCNCPoint4[4330] = {X 173.3257, Y 23.3717, Z -5.5000, A 0.000, B 0.000, C 0.000 }
gfCNCPoint4[4331] = {X 172.7810, Y 22.7015, Z -5.5000, A 0.000, B 0.000, C 0.000 }
gfCNCPoint4[4332] = {X 172.3776, Y 21.9378, Z -5.5000, A 0.000, B 0.000, C 0.000 }
gfCNCPoint4[4333] = {X 169.7664, Y 15.5423, Z -5.5000, A 0.000, B 0.000, C 0.000 }
gfCNCPoint4[4334] = {X 169.5125, Y 14.6752, Z -5.5000, A 0.000, B 0.000, C 0.000 }
gfCNCPoint4[4335] = {X 169.4412, Y 13.7745, Z -5.5000, A 0.000, B 0.000, C 0.000 }
gfCNCPoint4[4336] = {X 169.5553, Y 12.8782, Z -5.5000, A 0.000, B 0.000, C 0.000 }
gfCNCPoint4[4337] = {X 169.8501, Y 12.0241, Z -5.5000, A 0.000, B 0.000, C 0.000 }
gfCNCPoint4[4338] = {X 170.3131, Y 11.2482, Z -5.5000, A 0.000, B 0.000, C 0.000 }
gfCNCPoint4[4339] = {X 170.9249, Y 10.5833, Z -5.5000, A 0.000, B 0.000, C 0.000 }
gfCNCPoint4[4340] = {X 171.6596, Y 10.0573, Z -5.5000, A 0.000, B 0.000, C 0.000 }
gfCNCPoint4[4341] = {X 172.2916, Y 9.6970, Z -5.5000, A 0.000, B 0.000, C 0.000 }
gfCNCPoint4[4342] = {X 173.1775, Y 9.3226, Z -5.5000, A 0.000, B 0.000, C 0.000 }
gfCNCPoint4[4343] = {X 174.1236, Y 9.1496, Z -5.5000, A 0.000, B 0.000, C 0.000 }
gfCNCPoint4[4344] = {X 175.0846, Y 9.1864, Z -5.5000, A 0.000, B 0.000, C 0.000 }
gfCNCPoint4[4345] = {X 176.0147, Y 9.4310, Z -5.5000, A 0.000, B 0.000, C 0.000 }
gfCNCPoint4[4346] = {X 177.1120, Y 8.9641, Z -5.5000, A 0.000, B 0.000, C 0.000 }
gfCNCPoint4[4347] = {X 179.2948, Y 8.1608, Z -5.5000, A 0.000, B 0.000, C 0.000 }
gfCNCPoint4[4348] = {X 181.5465, Y 7.5780, Z -5.5000, A 0.000, B 0.000, C 0.000 }
gfCNCPoint4[4349] = {X 183.8450, Y 7.2215, Z -5.5000, A 0.000, B 0.000, C 0.000 }
gfCNCPoint4[4350] = {X 186.1675, Y 7.0949, Z -5.5000, A 0.000, B 0.000, C 0.000 }
gfCNCPoint4[4351] = {X 188.4911, Y 7.1993, Z -5.5000, A 0.000, B 0.000, C 0.000 }
gfCNCPoint4[4352] = {X 190.7928, Y 7.5337, Z -5.5000, A 0.000, B 0.000, C 0.000 }
gfCNCPoint4[4353] = {X 192.3783, Y 7.9242, Z -5.5000, A 0.000, B 0.000, C 0.000 }
gfCNCPoint4[4354] = {X 193.9195, Y 8.4633, Z -5.5000, A 0.000, B 0.000, C 0.000 }
gfCNCPoint4[4355] = {X 195.4027, Y 9.1462, Z -5.5000, A 0.000, B 0.000, C 0.000 }
gfCNCPoint4[4356] = {X 196.8144, Y 9.9666, Z -5.5000, A 0.000, B 0.000, C 0.000 }
gfCNCPoint4[4357] = {X 198.1419, Y 10.9173, Z -5.5000, A 0.000, B 0.000, C 0.000 }
gfCNCPoint4[4358] = {X 199.2087, Y 11.8667, Z -5.5000, A 0.000, B 0.000, C 0.000 }
gfCNCPoint4[4359] = {X 200.1658, Y 12.9264, Z -5.5000, A 0.000, B 0.000, C 0.000 }
gfCNCPoint4[4360] = {X 201.0020, Y 14.0840, Z -5.5000, A 0.000, B 0.000, C 0.000 }
gfCNCPoint4[4361] = {X 201.7072, Y 15.3258, Z -5.5000, A 0.000, B 0.000, C 0.000 }
gfCNCPoint4[4362] = {X 202.2731, Y 16.6369, Z -5.5000, A 0.000, B 0.000, C 0.000 }
gfCNCPoint4[4363] = {X 202.7492, Y 18.3014, Z -5.5000, A 0.000, B 0.000, C 0.000 }
gfCNCPoint4[4364] = {X 203.0318, Y 20.0095, Z -5.5000, A 0.000, B 0.000, C 0.000 }
gfCNCPoint4[4365] = {X 203.1170, Y 21.7387, Z -5.5000, A 0.000, B 0.000, C 0.000 }
gfCNCPoint4[4366] = {X 203.0038, Y 23.4663, Z -5.5000, A 0.000, B 0.000, C 0.000 }
gfCNCPoint4[4367] = {X 202.6936, Y 25.1696, Z -5.5000, A 0.000, B 0.000, C 0.000 }
gfCNCPoint4[4368] = {X 202.2588, Y 26.5986, Z -5.5000, A 0.000, B 0.000, C 0.000 }
gfCNCPoint4[4369] = {X 201.6467, Y 27.9611, Z -5.5000, A 0.000, B 0.000, C 0.000 }
gfCNCPoint4[4370] = {X 200.8670, Y 29.2351, Z -5.5000, A 0.000, B 0.000, C 0.000 }
gfCNCPoint4[4371] = {X 199.9322, Y 30.4001, Z -5.5000, A 0.000, B 0.000, C 0.000 }
gfCNCPoint4[4372] = {X 198.8575, Y 31.4374, Z -5.5000, A 0.000, B 0.000, C 0.000 }
gfCNCPoint4[4373] = {X 199.6405, Y 31.7992, Z -5.5000, A 0.000, B 0.000, C 0.000 }
gfCNCPoint4[4374] = {X 200.3379, Y 32.3068, Z -5.5000, A 0.000, B 0.000, C 0.000 }
gfCNCPoint4[4375] = {X 200.9229, Y 32.9406, Z -5.5000, A 0.000, B 0.000, C 0.000 }
gfCNCPoint4[4376] = {X 201.3730, Y 33.6764, Z -5.5000, A 0.000, B 0.000, C 0.000 }
gfCNCPoint4[4377] = {X 204.3942, Y 39.9182, Z -5.5000, A 0.000, B 0.000, C 0.000 }
gfCNCPoint4[4378] = {X 204.7207, Y 40.8441, Z -5.5000, A 0.000, B 0.000, C 0.000 }
gfCNCPoint4[4379] = {X 204.8337, Y 41.8194, Z -5.5000, A 0.000, B 0.000, C 0.000 }
gfCNCPoint4[4380] = {X 204.7276, Y 42.7955, Z -5.5000, A 0.000, B 0.000, C 0.000 }
gfCNCPoint4[4381] = {X 204.4078, Y 43.7238, Z -5.5000, A 0.000, B 0.000, C 0.000 }
gfCNCPoint4[4382] = {X 203.8900, Y 44.5580, Z -5.5000, A 0.000, B 0.000, C 0.000 }
gfCNCPoint4[4383] = {X 203.2002, Y 45.2567, Z -5.5000, A 0.000, B 0.000, C 0.000 }
gfCNCPoint4[4384] = {X 202.6640, Y 45.6902, Z -5.5000, A 0.000, B 0.000, C 0.000 }
gfCNCPoint4[4385] = {X 201.9527, Y 46.1595, Z -5.5000, A 0.000, B 0.000, C 0.000 }
gfCNCPoint4[4386] = {X 201.1644, Y 46.4832, Z -5.5000, A 0.000, B 0.000, C 0.000 }
gfCNCPoint4[4387] = {X 200.3286, Y 46.6493, Z -5.5000, A 0.000, B 0.000, C 0.000 }
gfCNCPoint4[4388] = {X 199.4764, Y 46.6516, Z -5.5000, A 0.000, B 0.000, C 0.000 }
gfCNCPoint4[4389] = {X 198.6397, Y 46.4900, Z -5.5000, A 0.000, B 0.000, C 0.000 }
gfCNCPoint4[4390] = {X 196.5324, Y 47.5866, Z -5.5000, A 0.000, B 0.000, C 0.000 }
gfCNCPoint4[4391] = {X 194.3411, Y 48.5038, Z -5.5000, A 0.000, B 0.000, C 0.000 }
gfCNCPoint4[4392] = {X 192.0811, Y 49.2352, Z -5.5000, A 0.000, B 0.000, C 0.000 }
gfCNCPoint4[4393] = {X 190.2776, Y 49.6708, Z -5.5000, A 0.000, B 0.000, C 0.000 }
gfCNCPoint4[4394] = {X 188.4443, Y 49.9564, Z -5.5000, A 0.000, B 0.000, C 0.000 }
gfCNCPoint4[4395] = {X 186.5937, Y 50.0898, Z -5.5000, A 0.000, B 0.000, C 0.000 }
gfCNCPoint4[4396] = {X 184.7384, Y 50.0702, Z -5.5000, A 0.000, B 0.000, C 0.000 }
gfCNCPoint4[4397] = {X 184.7136, Y 50.5496, Z -5.5000, A 0.000, B 0.000, C 0.000 }
gfCNCPoint4[4398] = {X 185.7092, Y 51.5029, Z -5.5000, A 0.000, B 0.000, C 0.000 }
gfCNCPoint4[4399] = {X 186.5593, Y 52.5880, Z -5.5000, A 0.000, B 0.000, C 0.000 }
gfCNCPoint4[4400] = {X 187.2466, Y 53.7828, Z -5.5000, A 0.000, B 0.000, C 0.000 }
gfCNCPoint4[4401] = {X 187.7797, Y 55.1346, Z -5.5000, A 0.000, B 0.000, C 0.000 }
gfCNCPoint4[4402] = {X 188.1044, Y 56.5510, Z -5.5000, A 0.000, B 0.000, C 0.000 }
gfCNCPoint4[4403] = {X 188.2135, Y 58.0000, Z -5.5000, A 0.000, B 0.000, C 0.000 }
gfCNCPoint4[4404] = {X 188.2132, Y 59.0140, Z -5.5000, A 0.000, B 0.000, C 0.000 }
gfCNCPoint4[4405] = {X 188.2026, Y 59.3924, Z -5.5000, A 0.000, B 0.000, C 0.000 }
gfCNCPoint4[4406] = {X 188.1773, Y 59.7701, Z -5.5000, A 0.000, B 0.000, C 0.000 }
gfCNCPoint4[4407] = {X 213.4312, Y 87.3333, Z -5.5000, A 0.000, B 0.000, C 0.000 }
gfCNCPoint4[4408] = {X 213.5228, Y 87.4315, Z -5.5000, A 0.000, B 0.000, C 0.000 }
gfCNCPoint4[4409] = {X 214.2178, Y 87.3790, Z -5.5000, A 0.000, B 0.000, C 0.000 }
gfCNCPoint4[4410] = {X 214.9136, Y 87.3375, Z -5.5000, A 0.000, B 0.000, C 0.000 }
gfCNCPoint4[4411] = {X 234.0911, Y 75.0518, Z -5.5000, A 0.000, B 0.000, C 0.000 }
gfCNCPoint4[4412] = {X 219.6589, Y 69.3883, Z -5.5000, A 0.000, B 0.000, C 0.000 }
gfCNCPoint4[4413] = {X 218.4694, Y 68.9881, Z -5.5000, A 0.000, B 0.000, C 0.000 }
gfCNCPoint4[4414] = {X 217.2417, Y 68.7269, Z -5.5000, A 0.000, B 0.000, C 0.000 }
gfCNCPoint4[4415] = {X 215.9923, Y 68.6081, Z -5.5000, A 0.000, B 0.000, C 0.000 }
gfCNCPoint4[4416] = {X 214.5221, Y 68.4436, Z -5.5000, A 0.000, B 0.000, C 0.000 }
gfCNCPoint4[4417] = {X 213.0942, Y 68.0569, Z -5.5000, A 0.000, B 0.000, C 0.000 }
gfCNCPoint4[4418] = {X 211.7419, Y 67.4572, Z -5.5000, A 0.000, B 0.000, C 0.000 }
gfCNCPoint4[4419] = {X 210.4967, Y 66.6584, Z -5.5000, A 0.000, B 0.000, C 0.000 }
gfCNCPoint4[4420] = {X 209.3878, Y 65.6793, Z -5.5000, A 0.000, B 0.000, C 0.000 }
gfCNCPoint4[4421] = {X 208.4411, Y 64.5426, Z -5.5000, A 0.000, B 0.000, C 0.000 }
gfCNCPoint4[4422] = {X 207.6786, Y 63.2749, Z -5.5000, A 0.000, B 0.000, C 0.000 }
gfCNCPoint4[4423] = {X 207.1182, Y 61.9058, Z -5.5000, A 0.000, B 0.000, C 0.000 }
gfCNCPoint4[4424] = {X 206.7730, Y 60.4673, Z -5.5000, A 0.000, B 0.000, C 0.000 }
gfCNCPoint4[4425] = {X 206.6510, Y 58.9930, Z -5.5000, A 0.000, B 0.000, C 0.000 }
gfCNCPoint4[4426] = {X 206.6508, Y 58.0000, Z -5.5000, A 0.000, B 0.000, C 0.000 }
gfCNCPoint4[4427] = {X 206.7577, Y 56.5655, Z -5.5000, A 0.000, B 0.000, C 0.000 }
gfCNCPoint4[4428] = {X 207.0759, Y 55.1628, Z -5.5000, A 0.000, B 0.000, C 0.000 }
gfCNCPoint4[4429] = {X 207.5986, Y 53.8226, Z -5.5000, A 0.000, B 0.000, C 0.000 }
gfCNCPoint4[4430] = {X 208.3140, Y 52.5747, Z -5.5000, A 0.000, B 0.000, C 0.000 }
gfCNCPoint4[4431] = {X 209.2065, Y 51.4466, Z -5.5000, A 0.000, B 0.000, C 0.000 }
gfCNCPoint4[4432] = {X 210.2563, Y 50.4632, Z -5.5000, A 0.000, B 0.000, C 0.000 }
gfCNCPoint4[4433] = {X 211.4402, Y 49.6463, Z -5.5000, A 0.000, B 0.000, C 0.000 }
gfCNCPoint4[4434] = {X 212.5893, Y 49.0723, Z -5.5000, A 0.000, B 0.000, C 0.000 }
gfCNCPoint4[4435] = {X 213.8042, Y 48.6556, Z -5.5000, A 0.000, B 0.000, C 0.000 }
gfCNCPoint4[4436] = {X 213.2578, Y 48.0874, Z -5.5000, A 0.000, B 0.000, C 0.000 }
gfCNCPoint4[4437] = {X 212.8100, Y 47.4386, Z -5.5000, A 0.000, B 0.000, C 0.000 }
gfCNCPoint4[4438] = {X 212.4725, Y 46.7262, Z -5.5000, A 0.000, B 0.000, C 0.000 }
gfCNCPoint4[4439] = {X 212.2401, Y 45.8965, Z -5.5000, A 0.000, B 0.000, C 0.000 }
gfCNCPoint4[4440] = {X 212.1572, Y 45.0389, Z -5.5000, A 0.000, B 0.000, C 0.000 }
gfCNCPoint4[4441] = {X 212.1570, Y 44.1949, Z -5.5000, A 0.000, B 0.000, C 0.000 }
gfCNCPoint4[4442] = {X 212.2383, Y 43.3144, Z -5.5000, A 0.000, B 0.000, C 0.000 }
gfCNCPoint4[4443] = {X 212.4794, Y 42.4638, Z -5.5000, A 0.000, B 0.000, C 0.000 }
gfCNCPoint4[4444] = {X 212.8721, Y 41.6716, Z -5.5000, A 0.000, B 0.000, C 0.000 }
gfCNCPoint4[4445] = {X 213.4033, Y 40.9647, Z -5.5000, A 0.000, B 0.000, C 0.000 }
gfCNCPoint4[4446] = {X 213.6818, Y 40.6575, Z -5.5000, A 0.000, B 0.000, C 0.000 }
gfCNCPoint4[4447] = {X 213.6845, Y 40.3041, Z -5.5000, A 0.000, B 0.000, C 0.000 }
gfCNCPoint4[4448] = {X 213.6845, Y 17.4645, Z -5.5000, A 0.000, B 0.000, C 0.000 }
gfCNCPoint4[4449] = {X 213.6792, Y 16.7696, Z -5.5000, A 0.000, B 0.000, C 0.000 }
gfCNCPoint4[4450] = {X 213.6790, Y 16.5189, Z -5.5000, A 0.000, B 0.000, C 0.000 }
gfCNCPoint4[4451] = {X 213.0400, Y 15.7777, Z -5.5000, A 0.000, B 0.000, C 0.000 }
gfCNCPoint4[4452] = {X 212.5617, Y 14.9238, Z -5.5000, A 0.000, B 0.000, C 0.000 }
gfCNCPoint4[4453] = {X 212.2635, Y 13.9917, Z -5.5000, A 0.000, B 0.000, C 0.000 }
gfCNCPoint4[4454] = {X 212.1572, Y 13.0188, Z -5.5000, A 0.000, B 0.000, C 0.000 }
gfCNCPoint4[4455] = {X 212.1570, Y 12.1868, Z -5.5000, A 0.000, B 0.000, C 0.000 }
gfCNCPoint4[4456] = {X 212.2436, Y 11.2717, Z -5.5000, A 0.000, B 0.000, C 0.000 }
gfCNCPoint4[4457] = {X 212.5002, Y 10.3891, Z -5.5000, A 0.000, B 0.000, C 0.000 }
gfCNCPoint4[4458] = {X 212.9449, Y 9.5280, Z -5.5000, A 0.000, B 0.000, C 0.000 }
gfCNCPoint4[4459] = {X 213.5510, Y 8.7718, Z -5.5000, A 0.000, B 0.000, C 0.000 }
gfCNCPoint4[4460] = {X 214.2946, Y 8.1503, Z -5.5000, A 0.000, B 0.000, C 0.000 }
gfCNCPoint4[4461] = {X 215.1464, Y 7.6879, Z -5.5000, A 0.000, B 0.000, C 0.000 }
gfCNCPoint4[4462] = {X 216.0727, Y 7.4030, Z -5.5000, A 0.000, B 0.000, C 0.000 }
gfCNCPoint4[4463] = {X 217.0370, Y 7.3068, Z -5.5000, A 0.000, B 0.000, C 0.000 }
gfCNCPoint4[4464] = {X 223.4805, Y 7.3068, Z -5.5000, A 0.000, B 0.000, C 0.000 }
gfCNCPoint4[4465] = {X 224.4448, Y 7.4030, Z -5.5000, A 0.000, B 0.000, C 0.000 }
gfCNCPoint4[4466] = {X 225.3711, Y 7.6879, Z -5.5000, A 0.000, B 0.000, C 0.000 }
gfCNCPoint4[4467] = {X 226.2229, Y 8.1503, Z -5.5000, A 0.000, B 0.000, C 0.000 }
gfCNCPoint4[4468] = {X 226.9665, Y 8.7718, Z -5.5000, A 0.000, B 0.000, C 0.000 }
gfCNCPoint4[4469] = {X 227.5726, Y 9.5280, Z -5.5000, A 0.000, B 0.000, C 0.000 }
gfCNCPoint4[4470] = {X 228.0173, Y 10.3891, Z -5.5000, A 0.000, B 0.000, C 0.000 }
gfCNCPoint4[4471] = {X 228.2739, Y 11.2717, Z -5.5000, A 0.000, B 0.000, C 0.000 }
gfCNCPoint4[4472] = {X 228.3605, Y 12.1868, Z -5.5000, A 0.000, B 0.000, C 0.000 }
gfCNCPoint4[4473] = {X 228.3603, Y 13.0237, Z -5.5000, A 0.000, B 0.000, C 0.000 }
gfCNCPoint4[4474] = {X 228.2529, Y 13.9970, Z -5.5000, A 0.000, B 0.000, C 0.000 }
gfCNCPoint4[4475] = {X 227.9534, Y 14.9292, Z -5.5000, A 0.000, B 0.000, C 0.000 }
gfCNCPoint4[4476] = {X 227.4739, Y 15.7829, Z -5.5000, A 0.000, B 0.000, C 0.000 }
gfCNCPoint4[4477] = {X 226.8336, Y 16.5236, Z -5.5000, A 0.000, B 0.000, C 0.000 }
gfCNCPoint4[4478] = {X 226.8345, Y 40.6640, Z -5.5000, A 0.000, B 0.000, C 0.000 }
gfCNCPoint4[4479] = {X 227.4745, Y 41.4049, Z -5.5000, A 0.000, B 0.000, C 0.000 }
gfCNCPoint4[4480] = {X 227.9538, Y 42.2585, Z -5.5000, A 0.000, B 0.000, C 0.000 }
gfCNCPoint4[4481] = {X 228.2531, Y 43.1907, Z -5.5000, A 0.000, B 0.000, C 0.000 }
gfCNCPoint4[4482] = {X 228.3603, Y 44.1638, Z -5.5000, A 0.000, B 0.000, C 0.000 }
gfCNCPoint4[4483] = {X 228.3605, Y 45.0000, Z -5.5000, A 0.000, B 0.000, C 0.000 }
gfCNCPoint4[4484] = {X 228.3507, Y 45.3090, Z -5.5000, A 0.000, B 0.000, C 0.000 }
gfCNCPoint4[4485] = {X 228.3214, Y 45.6167, Z -5.5000, A 0.000, B 0.000, C 0.000 }
gfCNCPoint4[4486] = {X 228.0910, Y 46.5992, Z -5.5000, A 0.000, B 0.000, C 0.000 }
gfCNCPoint4[4487] = {X 227.6635, Y 47.5134, Z -5.5000, A 0.000, B 0.000, C 0.000 }
gfCNCPoint4[4488] = {X 227.0571, Y 48.3200, Z -5.5000, A 0.000, B 0.000, C 0.000 }
gfCNCPoint4[4489] = {X 226.7053, Y 47.9934, Z -5.5000, A 0.000, B 0.000, C 0.000 }
gfCNCPoint4[4490] = {X 226.0261, Y 48.5889, Z -5.5000, A 0.000, B 0.000, C 0.000 }
gfCNCPoint4[4491] = {X 225.2396, Y 49.0331, Z -5.5000, A 0.000, B 0.000, C 0.000 }
gfCNCPoint4[4492] = {X 224.3790, Y 49.3073, Z -5.5000, A 0.000, B 0.000, C 0.000 }
gfCNCPoint4[4493] = {X 223.4805, Y 49.4000, Z -5.5000, A 0.000, B 0.000, C 0.000 }
gfCNCPoint4[4494] = {X 217.0370, Y 49.4000, Z -5.5000, A 0.000, B 0.000, C 0.000 }
gfCNCPoint4[4495] = {X 216.0579, Y 49.2897, Z -5.5000, A 0.000, B 0.000, C 0.000 }
gfCNCPoint4[4496] = {X 215.1279, Y 48.9643, Z -5.5000, A 0.000, B 0.000, C 0.000 }
gfCNCPoint4[4497] = {X 214.2937, Y 48.4400, Z -5.5000, A 0.000, B 0.000, C 0.000 }
gfCNCPoint4[4498] = {X 213.5969, Y 47.7433, Z -5.5000, A 0.000, B 0.000, C 0.000 }
gfCNCPoint4[4499] = {X 213.0727, Y 46.9091, Z -5.5000, A 0.000, B 0.000, C 0.000 }
gfCNCPoint4[4500] = {X 212.7473, Y 45.9791, Z -5.5000, A 0.000, B 0.000, C 0.000 }
gfCNCPoint4[4501] = {X 212.6370, Y 45.0000, Z -5.5000, A 0.000, B 0.000, C 0.000 }
gfCNCPoint4[4502] = {X 212.6370, Y 44.1949, Z -5.5000, A 0.000, B 0.000, C 0.000 }
gfCNCPoint4[4503] = {X 212.7102, Y 43.4023, Z -5.5000, A 0.000, B 0.000, C 0.000 }
gfCNCPoint4[4504] = {X 212.9272, Y 42.6365, Z -5.5000, A 0.000, B 0.000, C 0.000 }
gfCNCPoint4[4505] = {X 213.2808, Y 41.9234, Z -5.5000, A 0.000, B 0.000, C 0.000 }
gfCNCPoint4[4506] = {X 213.7589, Y 41.2871, Z -5.5000, A 0.000, B 0.000, C 0.000 }
gfCNCPoint4[4507] = {X 214.1604, Y 40.8442, Z -5.5000, A 0.000, B 0.000, C 0.000 }
gfCNCPoint4[4508] = {X 214.1645, Y 40.3060, Z -5.5000, A 0.000, B 0.000, C 0.000 }
gfCNCPoint4[4509] = {X 214.1645, Y 17.4626, Z -5.5000, A 0.000, B 0.000, C 0.000 }
gfCNCPoint4[4510] = {X 214.1592, Y 16.7691, Z -5.5000, A 0.000, B 0.000, C 0.000 }
gfCNCPoint4[4511] = {X 214.1588, Y 16.3060, Z -5.5000, A 0.000, B 0.000, C 0.000 }
gfCNCPoint4[4512] = {X 213.5165, Y 15.6173, Z -5.5000, A 0.000, B 0.000, C 0.000 }
gfCNCPoint4[4513] = {X 213.0355, Y 14.8077, Z -5.5000, A 0.000, B 0.000, C 0.000 }
gfCNCPoint4[4514] = {X 212.7378, Y 13.9143, Z -5.5000, A 0.000, B 0.000, C 0.000 }
gfCNCPoint4[4515] = {X 212.6370, Y 12.9780, Z -5.5000, A 0.000, B 0.000, C 0.000 }
gfCNCPoint4[4516] = {X 212.6370, Y 12.1868, Z -5.5000, A 0.000, B 0.000, C 0.000 }
gfCNCPoint4[4517] = {X 212.7473, Y 11.2077, Z -5.5000, A 0.000, B 0.000, C 0.000 }
gfCNCPoint4[4518] = {X 213.0728, Y 10.2777, Z -5.5000, A 0.000, B 0.000, C 0.000 }
gfCNCPoint4[4519] = {X 213.5970, Y 9.4435, Z -5.5000, A 0.000, B 0.000, C 0.000 }
gfCNCPoint4[4520] = {X 214.2937, Y 8.7468, Z -5.5000, A 0.000, B 0.000, C 0.000 }
gfCNCPoint4[4521] = {X 215.1279, Y 8.2226, Z -5.5000, A 0.000, B 0.000, C 0.000 }
gfCNCPoint4[4522] = {X 216.0579, Y 7.8971, Z -5.5000, A 0.000, B 0.000, C 0.000 }
gfCNCPoint4[4523] = {X 217.0370, Y 7.7868, Z -5.5000, A 0.000, B 0.000, C 0.000 }
gfCNCPoint4[4524] = {X 223.4805, Y 7.7868, Z -5.5000, A 0.000, B 0.000, C 0.000 }
gfCNCPoint4[4525] = {X 224.4596, Y 7.8971, Z -5.5000, A 0.000, B 0.000, C 0.000 }
gfCNCPoint4[4526] = {X 225.3896, Y 8.2226, Z -5.5000, A 0.000, B 0.000, C 0.000 }
gfCNCPoint4[4527] = {X 226.2238, Y 8.7468, Z -5.5000, A 0.000, B 0.000, C 0.000 }
gfCNCPoint4[4528] = {X 226.9205, Y 9.4435, Z -5.5000, A 0.000, B 0.000, C 0.000 }
gfCNCPoint4[4529] = {X 227.4447, Y 10.2777, Z -5.5000, A 0.000, B 0.000, C 0.000 }
gfCNCPoint4[4530] = {X 227.7702, Y 11.2077, Z -5.5000, A 0.000, B 0.000, C 0.000 }
gfCNCPoint4[4531] = {X 227.8805, Y 12.1868, Z -5.5000, A 0.000, B 0.000, C 0.000 }
gfCNCPoint4[4532] = {X 227.8802, Y 13.0233, Z -5.5000, A 0.000, B 0.000, C 0.000 }
gfCNCPoint4[4533] = {X 227.7720, Y 13.9492, Z -5.5000, A 0.000, B 0.000, C 0.000 }
gfCNCPoint4[4534] = {X 227.4711, Y 14.8314, Z -5.5000, A 0.000, B 0.000, C 0.000 }
gfCNCPoint4[4535] = {X 226.9911, Y 15.6305, Z -5.5000, A 0.000, B 0.000, C 0.000 }
gfCNCPoint4[4536] = {X 226.3535, Y 16.3105, Z -5.5000, A 0.000, B 0.000, C 0.000 }
gfCNCPoint4[4537] = {X 226.3545, Y 40.8771, Z -5.5000, A 0.000, B 0.000, C 0.000 }
gfCNCPoint4[4538] = {X 226.9985, Y 41.5661, Z -5.5000, A 0.000, B 0.000, C 0.000 }
gfCNCPoint4[4539] = {X 227.4808, Y 42.3766, Z -5.5000, A 0.000, B 0.000, C 0.000 }
gfCNCPoint4[4540] = {X 227.7794, Y 43.2712, Z -5.5000, A 0.000, B 0.000, C 0.000 }
gfCNCPoint4[4541] = {X 227.8805, Y 44.2089, Z -5.5000, A 0.000, B 0.000, C 0.000 }
gfCNCPoint4[4542] = {X 227.8805, Y 45.0000, Z -5.5000, A 0.000, B 0.000, C 0.000 }
gfCNCPoint4[4543] = {X 227.8037, Y 45.8182, Z -5.5000, A 0.000, B 0.000, C 0.000 }
gfCNCPoint4[4544] = {X 227.5762, Y 46.6079, Z -5.5000, A 0.000, B 0.000, C 0.000 }
gfCNCPoint4[4545] = {X 227.2057, Y 47.3415, Z -5.5000, A 0.000, B 0.000, C 0.000 }
gfCNCPoint4[4546] = {X 226.7053, Y 47.9934, Z -5.5000, A 0.000, B 0.000, C 0.000 }
gfCNCPoint4[4547] = {X 227.0571, Y 48.3200, Z -5.5000, A 0.000, B 0.000, C 0.000 }
gfCNCPoint4[4548] = {X 236.2309, Y 48.3200, Z -5.5000, A 0.000, B 0.000, C 0.000 }
gfCNCPoint4[4549] = {X 235.6245, Y 47.5134, Z -5.5000, A 0.000, B 0.000, C 0.000 }
gfCNCPoint4[4550] = {X 235.1970, Y 46.5992, Z -5.5000, A 0.000, B 0.000, C 0.000 }
gfCNCPoint4[4551] = {X 234.9666, Y 45.6167, Z -5.5000, A 0.000, B 0.000, C 0.000 }
gfCNCPoint4[4552] = {X 234.9373, Y 45.3090, Z -5.5000, A 0.000, B 0.000, C 0.000 }
gfCNCPoint4[4553] = {X 234.9275, Y 45.0000, Z -5.5000, A 0.000, B 0.000, C 0.000 }
gfCNCPoint4[4554] = {X 234.9275, Y 44.2089, Z -5.5000, A 0.000, B 0.000, C 0.000 }
gfCNCPoint4[4555] = {X 235.0194, Y 43.2661, Z -5.5000, A 0.000, B 0.000, C 0.000 }
gfCNCPoint4[4556] = {X 235.2918, Y 42.3588, Z -5.5000, A 0.000, B 0.000, C 0.000 }
gfCNCPoint4[4557] = {X 235.7342, Y 41.5212, Z -5.5000, A 0.000, B 0.000, C 0.000 }
gfCNCPoint4[4558] = {X 236.3302, Y 40.7849, Z -5.5000, A 0.000, B 0.000, C 0.000 }
gfCNCPoint4[4559] = {X 237.0572, Y 40.1776, Z -5.5000, A 0.000, B 0.000, C 0.000 }
gfCNCPoint4[4560] = {X 237.8878, Y 39.7222, Z -5.5000, A 0.000, B 0.000, C 0.000 }
gfCNCPoint4[4561] = {X 241.5462, Y 32.5613, Z -5.5000, A 0.000, B 0.000, C 0.000 }
gfCNCPoint4[4562] = {X 240.2117, Y 31.5585, Z -5.5000, A 0.000, B 0.000, C 0.000 }
gfCNCPoint4[4563] = {X 239.0309, Y 30.3786, Z -5.5000, A 0.000, B 0.000, C 0.000 }
gfCNCPoint4[4564] = {X 238.0272, Y 29.0448, Z -5.5000, A 0.000, B 0.000, C 0.000 }
gfCNCPoint4[4565] = {X 237.2203, Y 27.5835, Z -5.5000, A 0.000, B 0.000, C 0.000 }
gfCNCPoint4[4566] = {X 236.6262, Y 26.0235, Z -5.5000, A 0.000, B 0.000, C 0.000 }
gfCNCPoint4[4567] = {X 236.1911, Y 24.1499, Z -5.5000, A 0.000, B 0.000, C 0.000 }
gfCNCPoint4[4568] = {X 235.9692, Y 22.2393, Z -5.5000, A 0.000, B 0.000, C 0.000 }
gfCNCPoint4[4569] = {X 235.9633, Y 20.3159, Z -5.5000, A 0.000, B 0.000, C 0.000 }
gfCNCPoint4[4570] = {X 236.1735, Y 18.4039, Z -5.5000, A 0.000, B 0.000, C 0.000 }
gfCNCPoint4[4571] = {X 236.5972, Y 16.5277, Z -5.5000, A 0.000, B 0.000, C 0.000 }
gfCNCPoint4[4572] = {X 237.1166, Y 15.0571, Z -5.5000, A 0.000, B 0.000, C 0.000 }
gfCNCPoint4[4573] = {X 237.8163, Y 13.6632, Z -5.5000, A 0.000, B 0.000, C 0.000 }
gfCNCPoint4[4574] = {X 238.6853, Y 12.3681, Z -5.5000, A 0.000, B 0.000, C 0.000 }
gfCNCPoint4[4575] = {X 239.7100, Y 11.1923, Z -5.5000, A 0.000, B 0.000, C 0.000 }
gfCNCPoint4[4576] = {X 240.8743, Y 10.1540, Z -5.5000, A 0.000, B 0.000, C 0.000 }
gfCNCPoint4[4577] = {X 242.1597, Y 9.2700, Z -5.5000, A 0.000, B 0.000, C 0.000 }
gfCNCPoint4[4578] = {X 243.5459, Y 8.5543, Z -5.5000, A 0.000, B 0.000, C 0.000 }
gfCNCPoint4[4579] = {X 245.0109, Y 8.0182, Z -5.5000, A 0.000, B 0.000, C 0.000 }
gfCNCPoint4[4580] = {X 246.5316, Y 7.6701, Z -5.5000, A 0.000, B 0.000, C 0.000 }
gfCNCPoint4[4581] = {X 248.6761, Y 7.3927, Z -5.5000, A 0.000, B 0.000, C 0.000 }
gfCNCPoint4[4582] = {X 250.8369, Y 7.3102, Z -5.5000, A 0.000, B 0.000, C 0.000 }
gfCNCPoint4[4583] = {X 266.7608, Y 7.3102, Z -5.5000, A 0.000, B 0.000, C 0.000 }
gfCNCPoint4[4584] = {X 267.7191, Y 7.4117, Z -5.5000, A 0.000, B 0.000, C 0.000 }
gfCNCPoint4[4585] = {X 268.6389, Y 7.6994, Z -5.5000, A 0.000, B 0.000, C 0.000 }
gfCNCPoint4[4586] = {X 269.4842, Y 8.1621, Z -5.5000, A 0.000, B 0.000, C 0.000 }
gfCNCPoint4[4587] = {X 270.2222, Y 8.7819, Z -5.5000, A 0.000, B 0.000, C 0.000 }
gfCNCPoint4[4588] = {X 270.8240, Y 9.5345, Z -5.5000, A 0.000, B 0.000, C 0.000 }
gfCNCPoint4[4589] = {X 271.2664, Y 10.3907, Z -5.5000, A 0.000, B 0.000, C 0.000 }
gfCNCPoint4[4590] = {X 271.5234, Y 11.2719, Z -5.5000, A 0.000, B 0.000, C 0.000 }
gfCNCPoint4[4591] = {X 271.6110, Y 12.1856, Z -5.5000, A 0.000, B 0.000, C 0.000 }
gfCNCPoint4[4592] = {X 271.6108, Y 13.0237, Z -5.5000, A 0.000, B 0.000, C 0.000 }
gfCNCPoint4[4593] = {X 271.5128, Y 13.9524, Z -5.5000, A 0.000, B 0.000, C 0.000 }
gfCNCPoint4[4594] = {X 271.2396, Y 14.8453, Z -5.5000, A 0.000, B 0.000, C 0.000 }
gfCNCPoint4[4595] = {X 275.6743, Y 16.6820, Z -5.5000, A 0.000, B 0.000, C 0.000 }
gfCNCPoint4[4596] = {X 275.3128, Y 17.4564, Z -5.5000, A 0.000, B 0.000, C 0.000 }
gfCNCPoint4[4597] = {X 274.8843, Y 18.1959, Z -5.5000, A 0.000, B 0.000, C 0.000 }
gfCNCPoint4[4598] = {X 274.8842, Y 38.9907, Z -5.5000, A 0.000, B 0.000, C 0.000 }
gfCNCPoint4[4599] = {X 275.3140, Y 39.7328, Z -5.5000, A 0.000, B 0.000, C 0.000 }
gfCNCPoint4[4600] = {X 275.6765, Y 40.5100, Z -5.5000, A 0.000, B 0.000, C 0.000 }
gfCNCPoint4[4601] = {X 276.0375, Y 39.7356, Z -5.5000, A 0.000, B 0.000, C 0.000 }
gfCNCPoint4[4602] = {X 276.4650, Y 38.9959, Z -5.5000, A 0.000, B 0.000, C 0.000 }
gfCNCPoint4[4603] = {X 276.4646, Y 18.1963, Z -5.5000, A 0.000, B 0.000, C 0.000 }
gfCNCPoint4[4604] = {X 276.0360, Y 17.4566, Z -5.5000, A 0.000, B 0.000, C 0.000 }
gfCNCPoint4[4605] = {X 275.6743, Y 16.6820, Z -5.5000, A 0.000, B 0.000, C 0.000 }
gfCNCPoint4[4606] = {X 273.4570, Y 15.7637, Z -5.5000, A 0.000, B 0.000, C 0.000 }
gfCNCPoint4[4607] = {X 273.0266, Y 16.6337, Z -5.5000, A 0.000, B 0.000, C 0.000 }
gfCNCPoint4[4608] = {X 272.4843, Y 17.4387, Z -5.5000, A 0.000, B 0.000, C 0.000 }
gfCNCPoint4[4609] = {X 272.4842, Y 39.7479, Z -5.5000, A 0.000, B 0.000, C 0.000 }
gfCNCPoint4[4610] = {X 273.0276, Y 40.5548, Z -5.5000, A 0.000, B 0.000, C 0.000 }
gfCNCPoint4[4611] = {X 273.4586, Y 41.4270, Z -5.5000, A 0.000, B 0.000, C 0.000 }
gfCNCPoint4[4612] = {X 273.7588, Y 42.3092, Z -5.5000, A 0.000, B 0.000, C 0.000 }
gfCNCPoint4[4613] = {X 273.9439, Y 43.2224, Z -5.5000, A 0.000, B 0.000, C 0.000 }
gfCNCPoint4[4614] = {X 274.0108, Y 44.1519, Z -5.5000, A 0.000, B 0.000, C 0.000 }
gfCNCPoint4[4615] = {X 274.0110, Y 45.0000, Z -5.5000, A 0.000, B 0.000, C 0.000 }
gfCNCPoint4[4616] = {X 273.9884, Y 45.5734, Z -5.5000, A 0.000, B 0.000, C 0.000 }
gfCNCPoint4[4617] = {X 273.9207, Y 46.1433, Z -5.5000, A 0.000, B 0.000, C 0.000 }
gfCNCPoint4[4618] = {X 275.0713, Y 45.9760, Z -5.5000, A 0.000, B 0.000, C 0.000 }
gfCNCPoint4[4619] = {X 276.2327, Y 45.9200, Z -5.5000, A 0.000, B 0.000, C 0.000 }
gfCNCPoint4[4620] = {X 277.3960, Y 45.9200, Z -5.5000, A 0.000, B 0.000, C 0.000 }
gfCNCPoint4[4621] = {X 277.3539, Y 45.4857, Z -5.5000, A 0.000, B 0.000, C 0.000 }
gfCNCPoint4[4622] = {X 277.3378, Y 45.0498, Z -5.5000, A 0.000, B 0.000, C 0.000 }
gfCNCPoint4[4623] = {X 277.3377, Y 44.1989, Z -5.5000, A 0.000, B 0.000, C 0.000 }
gfCNCPoint4[4624] = {X 277.4028, Y 43.2536, Z -5.5000, A 0.000, B 0.000, C 0.000 }
gfCNCPoint4[4625] = {X 277.5893, Y 42.3246, Z -5.5000, A 0.000, B 0.000, C 0.000 }
gfCNCPoint4[4626] = {X 277.8942, Y 41.4275, Z -5.5000, A 0.000, B 0.000, C 0.000 }
gfCNCPoint4[4627] = {X 278.3239, Y 40.5569, Z -5.5000, A 0.000, B 0.000, C 0.000 }
gfCNCPoint4[4628] = {X 278.8650, Y 39.7509, Z -5.5000, A 0.000, B 0.000, C 0.000 }
gfCNCPoint4[4629] = {X 278.8646, Y 17.4391, Z -5.5000, A 0.000, B 0.000, C 0.000 }
gfCNCPoint4[4630] = {X 278.3222, Y 16.6339, Z -5.5000, A 0.000, B 0.000, C 0.000 }
gfCNCPoint4[4631] = {X 277.8917, Y 15.7637, Z -5.5000, A 0.000, B 0.000, C 0.000 }
gfCNCPoint4[4632] = {X 277.5902, Y 14.8788, Z -5.5000, A 0.000, B 0.000, C 0.000 }
gfCNCPoint4[4633] = {X 277.4046, Y 13.9627, Z -5.5000, A 0.000, B 0.000, C 0.000 }
gfCNCPoint4[4634] = {X 277.3379, Y 13.0303, Z -5.5000, A 0.000, B 0.000, C 0.000 }
gfCNCPoint4[4635] = {X 277.3377, Y 12.1868, Z -5.5000, A 0.000, B 0.000, C 0.000 }
gfCNCPoint4[4636] = {X 277.3952, Y 11.2737, Z -5.5000, A 0.000, B 0.000, C 0.000 }
gfCNCPoint4[4637] = {X 277.5667, Y 10.3750, Z -5.5000, A 0.000, B 0.000, C 0.000 }
gfCNCPoint4[4638] = {X 277.8497, Y 9.5049, Z -5.5000, A 0.000, B 0.000, C 0.000 }
gfCNCPoint4[4639] = {X 273.4969, Y 9.5049, Z -5.5000, A 0.000, B 0.000, C 0.000 }
gfCNCPoint4[4640] = {X 273.7802, Y 10.3734, Z -5.5000, A 0.000, B 0.000, C 0.000 }
gfCNCPoint4[4641] = {X 273.9524, Y 11.2705, Z -5.5000, A 0.000, B 0.000, C 0.000 }
gfCNCPoint4[4642] = {X 274.0110, Y 12.1822, Z -5.5000, A 0.000, B 0.000, C 0.000 }
gfCNCPoint4[4643] = {X 274.0107, Y 13.0462, Z -5.5000, A 0.000, B 0.000, C 0.000 }
gfCNCPoint4[4644] = {X 273.9427, Y 13.9732, Z -5.5000, A 0.000, B 0.000, C 0.000 }
gfCNCPoint4[4645] = {X 273.7571, Y 14.8840, Z -5.5000, A 0.000, B 0.000, C 0.000 }
gfCNCPoint4[4646] = {X 273.4570, Y 15.7637, Z -5.5000, A 0.000, B 0.000, C 0.000 }
gfCNCPoint4[4647] = {X 271.2396, Y 14.8453, Z -5.5000, A 0.000, B 0.000, C 0.000 }
gfCNCPoint4[4648] = {X 270.7505, Y 15.7453, Z -5.5000, A 0.000, B 0.000, C 0.000 }
gfCNCPoint4[4649] = {X 270.0843, Y 16.5234, Z -5.5000, A 0.000, B 0.000, C 0.000 }
gfCNCPoint4[4650] = {X 270.0842, Y 40.6632, Z -5.5000, A 0.000, B 0.000, C 0.000 }
gfCNCPoint4[4651] = {X 270.7245, Y 41.4040, Z -5.5000, A 0.000, B 0.000, C 0.000 }
gfCNCPoint4[4652] = {X 271.2040, Y 42.2578, Z -5.5000, A 0.000, B 0.000, C 0.000 }
gfCNCPoint4[4653] = {X 271.5035, Y 43.1900, Z -5.5000, A 0.000, B 0.000, C 0.000 }
gfCNCPoint4[4654] = {X 271.6108, Y 44.1633, Z -5.5000, A 0.000, B 0.000, C 0.000 }
gfCNCPoint4[4655] = {X 271.6110, Y 45.0000, Z -5.5000, A 0.000, B 0.000, C 0.000 }
gfCNCPoint4[4656] = {X 271.5959, Y 45.3844, Z -5.5000, A 0.000, B 0.000, C 0.000 }
gfCNCPoint4[4657] = {X 271.5505, Y 45.7664, Z -5.5000, A 0.000, B 0.000, C 0.000 }
gfCNCPoint4[4658] = {X 271.2989, Y 46.7171, Z -5.5000, A 0.000, B 0.000, C 0.000 }
gfCNCPoint4[4659] = {X 270.8619, Y 47.5982, Z -5.5000, A 0.000, B 0.000, C 0.000 }
gfCNCPoint4[4660] = {X 270.2571, Y 48.3736, Z -5.5000, A 0.000, B 0.000, C 0.000 }
gfCNCPoint4[4661] = {X 269.5090, Y 49.0121, Z -5.5000, A 0.000, B 0.000, C 0.000 }
gfCNCPoint4[4662] = {X 268.6482, Y 49.4876, Z -5.5000, A 0.000, B 0.000, C 0.000 }
gfCNCPoint4[4663] = {X 267.7095, Y 49.7809, Z -5.5000, A 0.000, B 0.000, C 0.000 }
gfCNCPoint4[4664] = {X 266.7310, Y 49.8800, Z -5.5000, A 0.000, B 0.000, C 0.000 }
gfCNCPoint4[4665] = {X 260.2876, Y 49.8800, Z -5.5000, A 0.000, B 0.000, C 0.000 }
gfCNCPoint4[4666] = {X 259.3711, Y 49.7932, Z -5.5000, A 0.000, B 0.000, C 0.000 }
gfCNCPoint4[4667] = {X 258.4873, Y 49.5358, Z -5.5000, A 0.000, B 0.000, C 0.000 }
gfCNCPoint4[4668] = {X 257.6675, Y 49.1170, Z -5.5000, A 0.000, B 0.000, C 0.000 }
gfCNCPoint4[4669] = {X 256.9410, Y 48.5517, Z -5.5000, A 0.000, B 0.000, C 0.000 }
gfCNCPoint4[4670] = {X 253.6492, Y 52.0452, Z -5.5000, A 0.000, B 0.000, C 0.000 }
gfCNCPoint4[4671] = {X 253.4932, Y 51.8948, Z -5.5000, A 0.000, B 0.000, C 0.000 }
gfCNCPoint4[4672] = {X 253.3406, Y 51.7410, Z -5.5000, A 0.000, B 0.000, C 0.000 }
gfCNCPoint4[4673] = {X 253.2764, Y 51.8066, Z -5.5000, A 0.000, B 0.000, C 0.000 }
gfCNCPoint4[4674] = {X 253.2116, Y 51.8715, Z -5.5000, A 0.000, B 0.000, C 0.000 }
gfCNCPoint4[4675] = {X 253.6492, Y 52.0452, Z -5.5000, A 0.000, B 0.000, C 0.000 }
gfCNCPoint4[4676] = {X 255.2951, Y 50.2985, Z -5.5000, A 0.000, B 0.000, C 0.000 }
gfCNCPoint4[4677] = {X 255.1778, Y 50.1854, Z -5.5000, A 0.000, B 0.000, C 0.000 }
gfCNCPoint4[4678] = {X 255.0630, Y 50.0697, Z -5.5000, A 0.000, B 0.000, C 0.000 }
gfCNCPoint4[4679] = {X 254.3405, Y 49.1989, Z -5.5000, A 0.000, B 0.000, C 0.000 }
gfCNCPoint4[4680] = {X 253.7617, Y 48.2267, Z -5.5000, A 0.000, B 0.000, C 0.000 }
gfCNCPoint4[4681] = {X 253.3406, Y 47.1766, Z -5.5000, A 0.000, B 0.000, C 0.000 }
gfCNCPoint4[4682] = {X 252.9194, Y 48.2267, Z -5.5000, A 0.000, B 0.000, C 0.000 }
gfCNCPoint4[4683] = {X 252.3406, Y 49.1989, Z -5.5000, A 0.000, B 0.000, C 0.000 }
gfCNCPoint4[4684] = {X 251.6182, Y 50.0697, Z -5.5000, A 0.000, B 0.000, C 0.000 }
gfCNCPoint4[4685] = {X 251.5699, Y 50.1190, Z -5.5000, A 0.000, B 0.000, C 0.000 }
gfCNCPoint4[4686] = {X 251.5211, Y 50.1678, Z -5.5000, A 0.000, B 0.000, C 0.000 }
gfCNCPoint4[4687] = {X 250.7152, Y 50.8585, Z -5.5000, A 0.000, B 0.000, C 0.000 }
gfCNCPoint4[4688] = {X 249.8174, Y 51.4246, Z -5.5000, A 0.000, B 0.000, C 0.000 }
gfCNCPoint4[4689] = {X 248.8468, Y 51.8542, Z -5.5000, A 0.000, B 0.000, C 0.000 }
gfCNCPoint4[4690] = {X 247.8241, Y 52.1381, Z -5.5000, A 0.000, B 0.000, C 0.000 }
gfCNCPoint4[4691] = {X 247.8928, Y 52.2637, Z -5.5000, A 0.000, B 0.000, C 0.000 }
gfCNCPoint4[4692] = {X 247.9601, Y 52.3902, Z -5.5000, A 0.000, B 0.000, C 0.000 }
gfCNCPoint4[4693] = {X 250.9677, Y 53.5630, Z -5.5000, A 0.000, B 0.000, C 0.000 }
gfCNCPoint4[4694] = {X 259.4019, Y 56.9107, Z -5.5000, A 0.000, B 0.000, C 0.000 }
gfCNCPoint4[4695] = {X 260.2873, Y 54.6800, Z -5.5000, A 0.000, B 0.000, C 0.000 }
gfCNCPoint4[4696] = {X 261.9957, Y 55.3581, Z -5.5000, A 0.000, B 0.000, C 0.000 }
gfCNCPoint4[4697] = {X 262.0630, Y 55.0182, Z -5.5000, A 0.000, B 0.000, C 0.000 }
gfCNCPoint4[4698] = {X 262.1384, Y 54.6800, Z -5.5000, A 0.000, B 0.000, C 0.000 }
gfCNCPoint4[4699] = {X 260.2873, Y 54.6800, Z -5.5000, A 0.000, B 0.000, C 0.000 }
gfCNCPoint4[4700] = {X 259.4019, Y 56.9107, Z -5.5000, A 0.000, B 0.000, C 0.000 }
gfCNCPoint4[4701] = {X 264.1528, Y 58.7964, Z -5.5000, A 0.000, B 0.000, C 0.000 }
gfCNCPoint4[4702] = {X 264.1527, Y 58.0000, Z -5.5000, A 0.000, B 0.000, C 0.000 }
gfCNCPoint4[4703] = {X 264.2035, Y 56.8933, Z -5.5000, A 0.000, B 0.000, C 0.000 }
gfCNCPoint4[4704] = {X 264.3555, Y 55.7960, Z -5.5000, A 0.000, B 0.000, C 0.000 }
gfCNCPoint4[4705] = {X 264.4116, Y 55.5124, Z -5.5000, A 0.000, B 0.000, C 0.000 }
gfCNCPoint4[4706] = {X 264.4745, Y 55.2303, Z -5.5000, A 0.000, B 0.000, C 0.000 }
gfCNCPoint4[4707] = {X 264.9369, Y 53.7185, Z -5.5000, A 0.000, B 0.000, C 0.000 }
gfCNCPoint4[4708] = {X 265.5928, Y 52.2800, Z -5.5000, A 0.000, B 0.000, C 0.000 }
gfCNCPoint4[4709] = {X 260.2876, Y 52.2800, Z -5.5000, A 0.000, B 0.000, C 0.000 }
gfCNCPoint4[4710] = {X 259.1915, Y 52.1970, Z -5.5000, A 0.000, B 0.000, C 0.000 }
gfCNCPoint4[4711] = {X 258.1204, Y 51.9500, Z -5.5000, A 0.000, B 0.000, C 0.000 }
gfCNCPoint4[4712] = {X 257.0987, Y 51.5444, Z -5.5000, A 0.000, B 0.000, C 0.000 }
gfCNCPoint4[4713] = {X 256.1497, Y 50.9897, Z -5.5000, A 0.000, B 0.000, C 0.000 }
gfCNCPoint4[4714] = {X 255.2951, Y 50.2985, Z -5.5000, A 0.000, B 0.000, C 0.000 }
gfCNCPoint4[4715] = {X 256.9410, Y 48.5517, Z -5.5000, A 0.000, B 0.000, C 0.000 }
gfCNCPoint4[4716] = {X 256.3869, Y 47.9324, Z -5.5000, A 0.000, B 0.000, C 0.000 }
gfCNCPoint4[4717] = {X 255.9459, Y 47.2280, Z -5.5000, A 0.000, B 0.000, C 0.000 }
gfCNCPoint4[4718] = {X 255.6308, Y 46.4590, Z -5.5000, A 0.000, B 0.000, C 0.000 }
gfCNCPoint4[4719] = {X 255.4666, Y 45.7568, Z -5.5000, A 0.000, B 0.000, C 0.000 }
gfCNCPoint4[4720] = {X 255.4077, Y 45.0380, Z -5.5000, A 0.000, B 0.000, C 0.000 }
gfCNCPoint4[4721] = {X 255.4080, Y 44.1417, Z -5.5000, A 0.000, B 0.000, C 0.000 }
gfCNCPoint4[4722] = {X 255.5183, Y 43.1751, Z -5.5000, A 0.000, B 0.000, C 0.000 }
gfCNCPoint4[4723] = {X 255.8181, Y 42.2497, Z -5.5000, A 0.000, B 0.000, C 0.000 }
gfCNCPoint4[4724] = {X 256.2955, Y 41.4021, Z -5.5000, A 0.000, B 0.000, C 0.000 }
gfCNCPoint4[4725] = {X 256.9315, Y 40.6660, Z -5.5000, A 0.000, B 0.000, C 0.000 }
gfCNCPoint4[4726] = {X 256.9315, Y 35.0338, Z -5.5000, A 0.000, B 0.000, C 0.000 }
gfCNCPoint4[4727] = {X 255.1100, Y 35.0338, Z -5.5000, A 0.000, B 0.000, C 0.000 }
gfCNCPoint4[4728] = {X 251.0866, Y 42.8709, Z -5.5000, A 0.000, B 0.000, C 0.000 }
gfCNCPoint4[4729] = {X 251.2237, Y 43.5129, Z -5.5000, A 0.000, B 0.000, C 0.000 }
gfCNCPoint4[4730] = {X 251.2734, Y 44.1675, Z -5.5000, A 0.000, B 0.000, C 0.000 }
gfCNCPoint4[4731] = {X 251.2736, Y 45.0000, Z -5.5000, A 0.000, B 0.000, C 0.000 }
gfCNCPoint4[4732] = {X 251.2174, Y 45.7380, Z -5.5000, A 0.000, B 0.000, C 0.000 }
gfCNCPoint4[4733] = {X 251.0503, Y 46.4590, Z -5.5000, A 0.000, B 0.000, C 0.000 }
gfCNCPoint4[4734] = {X 250.6346, Y 47.4142, Z -5.5000, A 0.000, B 0.000, C 0.000 }
gfCNCPoint4[4735] = {X 250.0255, Y 48.2593, Z -5.5000, A 0.000, B 0.000, C 0.000 }
gfCNCPoint4[4736] = {X 249.2510, Y 48.9560, Z -5.5000, A 0.000, B 0.000, C 0.000 }
gfCNCPoint4[4737] = {X 248.3462, Y 49.4723, Z -5.5000, A 0.000, B 0.000, C 0.000 }
gfCNCPoint4[4738] = {X 247.3525, Y 49.7849, Z -5.5000, A 0.000, B 0.000, C 0.000 }
gfCNCPoint4[4739] = {X 246.8754, Y 49.8562, Z -5.5000, A 0.000, B 0.000, C 0.000 }
gfCNCPoint4[4740] = {X 246.3936, Y 49.8800, Z -5.5000, A 0.000, B 0.000, C 0.000 }
gfCNCPoint4[4741] = {X 242.5312, Y 49.8800, Z -5.5000, A 0.000, B 0.000, C 0.000 }
gfCNCPoint4[4742] = {X 242.5312, Y 49.4000, Z -5.5000, A 0.000, B 0.000, C 0.000 }
gfCNCPoint4[4743] = {X 239.8075, Y 49.4000, Z -5.5000, A 0.000, B 0.000, C 0.000 }
gfCNCPoint4[4744] = {X 238.8284, Y 49.2897, Z -5.5000, A 0.000, B 0.000, C 0.000 }
gfCNCPoint4[4745] = {X 237.8984, Y 48.9643, Z -5.5000, A 0.000, B 0.000, C 0.000 }
gfCNCPoint4[4746] = {X 237.0641, Y 48.4401, Z -5.5000, A 0.000, B 0.000, C 0.000 }
gfCNCPoint4[4747] = {X 236.3674, Y 47.7434, Z -5.5000, A 0.000, B 0.000, C 0.000 }
gfCNCPoint4[4748] = {X 235.8432, Y 46.9091, Z -5.5000, A 0.000, B 0.000, C 0.000 }
gfCNCPoint4[4749] = {X 235.5178, Y 45.9791, Z -5.5000, A 0.000, B 0.000, C 0.000 }
gfCNCPoint4[4750] = {X 235.4075, Y 45.0000, Z -5.5000, A 0.000, B 0.000, C 0.000 }
gfCNCPoint4[4751] = {X 235.4079, Y 44.1483, Z -5.5000, A 0.000, B 0.000, C 0.000 }
gfCNCPoint4[4752] = {X 235.5063, Y 43.2816, Z -5.5000, A 0.000, B 0.000, C 0.000 }
gfCNCPoint4[4753] = {X 235.7737, Y 42.4514, Z -5.5000, A 0.000, B 0.000, C 0.000 }
gfCNCPoint4[4754] = {X 236.1996, Y 41.6903, Z -5.5000, A 0.000, B 0.000, C 0.000 }
gfCNCPoint4[4755] = {X 236.7672, Y 41.0281, Z -5.5000, A 0.000, B 0.000, C 0.000 }
gfCNCPoint4[4756] = {X 237.4544, Y 40.4909, Z -5.5000, A 0.000, B 0.000, C 0.000 }
gfCNCPoint4[4757] = {X 238.2339, Y 40.0998, Z -5.5000, A 0.000, B 0.000, C 0.000 }
gfCNCPoint4[4758] = {X 242.1746, Y 32.3863, Z -5.5000, A 0.000, B 0.000, C 0.000 }
gfCNCPoint4[4759] = {X 241.0110, Y 31.5938, Z -5.5000, A 0.000, B 0.000, C 0.000 }
gfCNCPoint4[4760] = {X 239.9540, Y 30.6640, Z -5.5000, A 0.000, B 0.000, C 0.000 }
gfCNCPoint4[4761] = {X 239.0197, Y 29.6109, Z -5.5000, A 0.000, B 0.000, C 0.000 }
gfCNCPoint4[4762] = {X 238.2223, Y 28.4507, Z -5.5000, A 0.000, B 0.000, C 0.000 }
gfCNCPoint4[4763] = {X 237.5739, Y 27.2010, Z -5.5000, A 0.000, B 0.000, C 0.000 }
gfCNCPoint4[4764] = {X 237.0846, Y 25.8809, Z -5.5000, A 0.000, B 0.000, C 0.000 }
gfCNCPoint4[4765] = {X 236.6628, Y 24.0613, Z -5.5000, A 0.000, B 0.000, C 0.000 }
gfCNCPoint4[4766] = {X 236.4480, Y 22.2057, Z -5.5000, A 0.000, B 0.000, C 0.000 }
gfCNCPoint4[4767] = {X 236.4428, Y 20.3378, Z -5.5000, A 0.000, B 0.000, C 0.000 }
gfCNCPoint4[4768] = {X 236.6473, Y 18.4811, Z -5.5000, A 0.000, B 0.000, C 0.000 }
gfCNCPoint4[4769] = {X 237.0589, Y 16.6591, Z -5.5000, A 0.000, B 0.000, C 0.000 }
gfCNCPoint4[4770] = {X 237.6331, Y 15.0728, Z -5.5000, A 0.000, B 0.000, C 0.000 }
gfCNCPoint4[4771] = {X 238.4254, Y 13.5834, Z -5.5000, A 0.000, B 0.000, C 0.000 }
gfCNCPoint4[4772] = {X 239.4199, Y 12.2206, Z -5.5000, A 0.000, B 0.000, C 0.000 }
gfCNCPoint4[4773] = {X 240.5967, Y 11.0118, Z -5.5000, A 0.000, B 0.000, C 0.000 }
gfCNCPoint4[4774] = {X 241.9323, Y 9.9810, Z -5.5000, A 0.000, B 0.000, C 0.000 }
gfCNCPoint4[4775] = {X 243.3999, Y 9.1490, Z -5.5000, A 0.000, B 0.000, C 0.000 }
gfCNCPoint4[4776] = {X 244.9703, Y 8.5323, Z -5.5000, A 0.000, B 0.000, C 0.000 }
gfCNCPoint4[4777] = {X 246.6119, Y 8.1434, Z -5.5000, A 0.000, B 0.000, C 0.000 }
gfCNCPoint4[4778] = {X 248.7155, Y 7.8711, Z -5.5000, A 0.000, B 0.000, C 0.000 }
gfCNCPoint4[4779] = {X 250.8351, Y 7.7902, Z -5.5000, A 0.000, B 0.000, C 0.000 }
gfCNCPoint4[4780] = {X 266.7640, Y 7.7902, Z -5.5000, A 0.000, B 0.000, C 0.000 }
gfCNCPoint4[4781] = {X 267.7369, Y 7.9071, Z -5.5000, A 0.000, B 0.000, C 0.000 }
gfCNCPoint4[4782] = {X 268.6599, Y 8.2363, Z -5.5000, A 0.000, B 0.000, C 0.000 }
gfCNCPoint4[4783] = {X 269.4872, Y 8.7616, Z -5.5000, A 0.000, B 0.000, C 0.000 }
gfCNCPoint4[4784] = {X 270.1778, Y 9.4568, Z -5.5000, A 0.000, B 0.000, C 0.000 }
gfCNCPoint4[4785] = {X 270.6975, Y 10.2875, Z -5.5000, A 0.000, B 0.000, C 0.000 }
gfCNCPoint4[4786] = {X 271.0206, Y 11.2126, Z -5.5000, A 0.000, B 0.000, C 0.000 }
gfCNCPoint4[4787] = {X 271.1310, Y 12.1863, Z -5.5000, A 0.000, B 0.000, C 0.000 }
gfCNCPoint4[4788] = {X 271.1308, Y 13.0233, Z -5.5000, A 0.000, B 0.000, C 0.000 }
gfCNCPoint4[4789] = {X 271.0225, Y 13.9491, Z -5.5000, A 0.000, B 0.000, C 0.000 }
gfCNCPoint4[4790] = {X 270.7217, Y 14.8313, Z -5.5000, A 0.000, B 0.000, C 0.000 }
gfCNCPoint4[4791] = {X 270.2418, Y 15.6303, Z -5.5000, A 0.000, B 0.000, C 0.000 }
gfCNCPoint4[4792] = {X 269.6043, Y 16.3103, Z -5.5000, A 0.000, B 0.000, C 0.000 }
gfCNCPoint4[4793] = {X 269.6042, Y 40.8764, Z -5.5000, A 0.000, B 0.000, C 0.000 }
gfCNCPoint4[4794] = {X 270.2485, Y 41.5654, Z -5.5000, A 0.000, B 0.000, C 0.000 }
gfCNCPoint4[4795] = {X 270.7312, Y 42.3760, Z -5.5000, A 0.000, B 0.000, C 0.000 }
gfCNCPoint4[4796] = {X 271.0299, Y 43.2709, Z -5.5000, A 0.000, B 0.000, C 0.000 }
gfCNCPoint4[4797] = {X 271.1310, Y 44.2089, Z -5.5000, A 0.000, B 0.000, C 0.000 }
gfCNCPoint4[4798] = {X 271.1310, Y 45.0000, Z -5.5000, A 0.000, B 0.000, C 0.000 }
gfCNCPoint4[4799] = {X 271.0207, Y 45.9791, Z -5.5000, A 0.000, B 0.000, C 0.000 }
gfCNCPoint4[4800] = {X 270.6953, Y 46.9091, Z -5.5000, A 0.000, B 0.000, C 0.000 }
gfCNCPoint4[4801] = {X 270.1711, Y 47.7434, Z -5.5000, A 0.000, B 0.000, C 0.000 }
gfCNCPoint4[4802] = {X 269.4744, Y 48.4401, Z -5.5000, A 0.000, B 0.000, C 0.000 }
gfCNCPoint4[4803] = {X 268.6401, Y 48.9643, Z -5.5000, A 0.000, B 0.000, C 0.000 }
gfCNCPoint4[4804] = {X 267.7101, Y 49.2897, Z -5.5000, A 0.000, B 0.000, C 0.000 }
gfCNCPoint4[4805] = {X 266.7310, Y 49.4000, Z -5.5000, A 0.000, B 0.000, C 0.000 }
gfCNCPoint4[4806] = {X 260.2876, Y 49.4000, Z -5.5000, A 0.000, B 0.000, C 0.000 }
gfCNCPoint4[4807] = {X 259.3085, Y 49.2897, Z -5.5000, A 0.000, B 0.000, C 0.000 }
gfCNCPoint4[4808] = {X 258.3785, Y 48.9643, Z -5.5000, A 0.000, B 0.000, C 0.000 }
gfCNCPoint4[4809] = {X 257.5442, Y 48.4400, Z -5.5000, A 0.000, B 0.000, C 0.000 }
gfCNCPoint4[4810] = {X 256.8475, Y 47.7433, Z -5.5000, A 0.000, B 0.000, C 0.000 }
gfCNCPoint4[4811] = {X 256.3233, Y 46.9091, Z -5.5000, A 0.000, B 0.000, C 0.000 }
gfCNCPoint4[4812] = {X 255.9979, Y 45.9791, Z -5.5000, A 0.000, B 0.000, C 0.000 }
gfCNCPoint4[4813] = {X 255.8876, Y 45.0000, Z -5.5000, A 0.000, B 0.000, C 0.000 }
gfCNCPoint4[4814] = {X 255.8880, Y 44.1483, Z -5.5000, A 0.000, B 0.000, C 0.000 }
gfCNCPoint4[4815] = {X 255.9984, Y 43.2275, Z -5.5000, A 0.000, B 0.000, C 0.000 }
gfCNCPoint4[4816] = {X 256.2993, Y 42.3503, Z -5.5000, A 0.000, B 0.000, C 0.000 }
gfCNCPoint4[4817] = {X 256.7775, Y 41.5556, Z -5.5000, A 0.000, B 0.000, C 0.000 }
gfCNCPoint4[4818] = {X 257.4115, Y 40.8789, Z -5.5000, A 0.000, B 0.000, C 0.000 }
gfCNCPoint4[4819] = {X 257.4115, Y 34.5538, Z -5.5000, A 0.000, B 0.000, C 0.000 }
gfCNCPoint4[4820] = {X 254.8169, Y 34.5538, Z -5.5000, A 0.000, B 0.000, C 0.000 }
gfCNCPoint4[4821] = {X 250.5704, Y 42.8254, Z -5.5000, A 0.000, B 0.000, C 0.000 }
gfCNCPoint4[4822] = {X 250.7374, Y 43.5082, Z -5.5000, A 0.000, B 0.000, C 0.000 }
gfCNCPoint4[4823] = {X 250.7936, Y 44.2089, Z -5.5000, A 0.000, B 0.000, C 0.000 }
gfCNCPoint4[4824] = {X 250.7936, Y 45.0000, Z -5.5000, A 0.000, B 0.000, C 0.000 }
gfCNCPoint4[4825] = {X 250.6832, Y 45.9791, Z -5.5000, A 0.000, B 0.000, C 0.000 }
gfCNCPoint4[4826] = {X 250.3578, Y 46.9091, Z -5.5000, A 0.000, B 0.000, C 0.000 }
gfCNCPoint4[4827] = {X 249.8336, Y 47.7434, Z -5.5000, A 0.000, B 0.000, C 0.000 }
gfCNCPoint4[4828] = {X 249.1369, Y 48.4401, Z -5.5000, A 0.000, B 0.000, C 0.000 }
gfCNCPoint4[4829] = {X 248.3026, Y 48.9643, Z -5.5000, A 0.000, B 0.000, C 0.000 }
gfCNCPoint4[4830] = {X 247.3727, Y 49.2897, Z -5.5000, A 0.000, B 0.000, C 0.000 }
gfCNCPoint4[4831] = {X 246.3936, Y 49.4000, Z -5.5000, A 0.000, B 0.000, C 0.000 }
gfCNCPoint4[4832] = {X 242.5312, Y 49.4000, Z -5.5000, A 0.000, B 0.000, C 0.000 }
gfCNCPoint4[4833] = {X 242.5312, Y 49.8800, Z -5.5000, A 0.000, B 0.000, C 0.000 }
gfCNCPoint4[4834] = {X 243.4812, Y 50.5824, Z -5.5000, A 0.000, B 0.000, C 0.000 }
gfCNCPoint4[4835] = {X 244.3384, Y 51.3953, Z -5.5000, A 0.000, B 0.000, C 0.000 }
gfCNCPoint4[4836] = {X 245.0903, Y 52.3066, Z -5.5000, A 0.000, B 0.000, C 0.000 }
gfCNCPoint4[4837] = {X 245.7256, Y 53.3027, Z -5.5000, A 0.000, B 0.000, C 0.000 }
gfCNCPoint4[4838] = {X 245.9755, Y 53.7843, Z -5.5000, A 0.000, B 0.000, C 0.000 }
gfCNCPoint4[4839] = {X 246.1980, Y 54.2791, Z -5.5000, A 0.000, B 0.000, C 0.000 }
gfCNCPoint4[4840] = {X 250.0857, Y 55.7950, Z -5.5000, A 0.000, B 0.000, C 0.000 }
gfCNCPoint4[4841] = {X 267.2822, Y 62.6207, Z -5.5000, A 0.000, B 0.000, C 0.000 }
gfCNCPoint4[4842] = {X 266.8843, Y 61.4460, Z -5.5000, A 0.000, B 0.000, C 0.000 }
gfCNCPoint4[4843] = {X 266.6398, Y 60.2302, Z -5.5000, A 0.000, B 0.000, C 0.000 }
gfCNCPoint4[4844] = {X 266.5529, Y 58.9930, Z -5.5000, A 0.000, B 0.000, C 0.000 }
gfCNCPoint4[4845] = {X 266.5527, Y 58.0000, Z -5.5000, A 0.000, B 0.000, C 0.000 }
